SPLINE
SPL {X  -153.420, Y  +337.122, Z    +0.000, E1  +333.501, E3 -305002.639}
SPL {X  -157.288, Y  +353.220, Z    +0.000, E1  +341.134, E3 -305014.684}
SPL {X  -159.049, Y  +365.172, Z    +0.000, E1  +347.392, E3 -305020.238}
SPL {X  -159.749, Y  +373.719, Z    +0.000, E1  +352.250, E3 -305022.858}
SPL {X  -159.988, Y  +381.741, Z    +0.000, E1  +357.172, E3 -305024.333}
SPL {X  -159.990, Y  +387.352, Z    +0.000, E1  +361.387, E3 -305025.035}
SPL {X  -159.990, Y  +391.188, Z    +0.000, E1  +365.082, E3 -305025.576}
SPL {X  -159.990, Y  +395.106, Z    +0.000, E1  +369.154, E3 -305026.317}
SPL {X  -159.990, Y  +400.303, Z    +0.000, E1  +374.927, E3 -305027.638}
SPL {X  -159.990, Y  +408.423, Z    +0.000, E1  +383.302, E3 -305030.717}
SPL {X  -159.990, Y  +438.418, Z    +0.000, E1  +401.067, E3 -305052.290}
SPL {X  -159.990, Y  +482.913, Z    +0.000, E1  +407.036, E3 -305111.644}
SPL {X  -159.990, Y  +489.230, Z    +0.000, E1  +407.019, E3 -305124.156}
SPL {X  -159.990, Y  +495.241, Z    +0.000, E1  +407.026, E3 -305136.035}
SPL {X  -159.990, Y  +501.001, Z    +0.000, E1  +407.020, E3 -305147.412}
SPL {X  -159.990, Y  +506.758, Z    +0.000, E1  +407.038, E3 -305158.758}
SPL {X  -159.990, Y  +512.807, Z    +0.000, E1  +407.022, E3 -305170.749}
SPL {X  -159.990, Y  +518.043, Z    +0.000, E1  +407.016, E3 -305181.127}
SPL {X  -159.990, Y  +523.058, Z    +0.000, E1  +407.015, E3 -305191.042}
SPL {X  -159.990, Y  +527.746, Z    +0.000, E1  +407.012, E3 -305200.316}
SPL {X  -159.990, Y  +533.771, Z    +0.000, E1  +407.034, E3 -305212.201}
SPL {X  -159.990, Y  +542.379, Z    +0.000, E1  +407.067, E3 -305229.170}
SPL {X  -159.990, Y  +549.846, Z    +0.000, E1  +407.016, E3 -305244.016}
SPL {X  -159.990, Y  +554.843, Z    +0.000, E1  +407.014, E3 -305253.894}
SPL {X  -159.990, Y  +560.453, Z    +0.000, E1  +407.023, E3 -305264.977}
SPL {X  -159.990, Y  +566.612, Z    +0.000, E1  +407.022, E3 -305277.159}
SPL {X  -159.990, Y  +572.901, Z    +0.000, E1  +407.028, E3 -305289.571}
SPL {X  -159.990, Y  +578.640, Z    +0.000, E1  +407.021, E3 -305300.922}
SPL {X  -159.990, Y  +583.515, Z    +0.000, E1  +407.019, E3 -305310.562}
SPL {X  -159.990, Y  +589.675, Z    +0.000, E1  +407.042, E3 -305322.700}
SPL {X  -159.990, Y  +596.627, Z    +0.000, E1  +407.034, E3 -305336.440}
SPL {X  -159.990, Y  +602.039, Z    +0.000, E1  +407.021, E3 -305347.147}
SPL {X  -159.990, Y  +607.106, Z    +0.000, E1  +407.028, E3 -305357.154}
SPL {X  -159.990, Y  +612.418, Z    +0.000, E1  +407.023, E3 -305367.665}
SPL {X  -159.990, Y  +618.496, Z    +0.000, E1  +407.049, E3 -305379.632}
SPL {X  -159.990, Y  +624.357, Z    +0.000, E1  +407.020, E3 -305391.258}
SPL {X  -159.990, Y  +629.711, Z    +0.000, E1  +407.034, E3 -305401.827}
SPL {X  -159.990, Y  +635.041, Z    +0.000, E1  +407.022, E3 -305412.372}
SPL {X  -159.990, Y  +639.998, Z    +0.000, E1  +407.027, E3 -305422.164}
SPL {X  -159.990, Y  +646.188, Z    +0.000, E1  +407.041, E3 -305434.390}
SPL {X  -159.990, Y  +652.067, Z    +0.000, E1  +407.023, E3 -305446.026}
SPL {X  -159.990, Y  +657.109, Z    +0.000, E1  +407.025, E3 -305456.005}
SPL {X  -159.990, Y  +662.651, Z    +0.000, E1  +407.027, E3 -305466.961}
SPL {X  -159.990, Y  +668.015, Z    +0.000, E1  +407.025, E3 -305477.561}
SPL {X  -159.972, Y  +673.909, Z    +0.000, E1  +407.029, E3 -305489.226}
SPL {X  -159.776, Y  +679.772, Z    +0.000, E1  +406.992, E3 -305501.027}
SPL {X  -159.384, Y  +685.411, Z    +0.000, E1  +406.921, E3 -305512.589}
SPL {X  -158.839, Y  +690.657, Z    +0.000, E1  +406.819, E3 -305523.543}
SPL {X  -157.875, Y  +697.431, Z    +0.000, E1  +406.688, E3 -305537.882}
SPL {X  -156.719, Y  +703.686, Z    +0.000, E1  +406.438, E3 -305551.492}
SPL {X  -155.778, Y  +707.970, Z    +0.000, E1  +406.262, E3 -305560.966}
SPL {X  -154.419, Y  +713.351, Z    +0.000, E1  +406.025, E3 -305572.998}
SPL {X  -152.913, Y  +718.557, Z    +0.000, E1  +405.729, E3 -305584.850}
SPL {X  -151.262, Y  +723.621, Z    +0.000, E1  +405.429, E3 -305596.516}
SPL {X  -149.074, Y  +729.584, Z    +0.000, E1  +405.040, E3 -305610.445}
SPL {X  -142.577, Y  +744.086, Z    +0.000, E1  +400.686, E3 -305676.651}
ENDSPLINE

SPLINE
SPL {X  -152.566, Y  +719.671, Z    +0.000, E1  +387.682, E3 -305747.122}
SPL {X  -158.253, Y  +695.011, Z    +0.000, E1  +375.913, E3 -305763.793}
SPL {X  -159.486, Y  +684.192, Z    +0.000, E1  +369.965, E3 -305767.740}
SPL {X  -159.898, Y  +676.924, Z    +0.000, E1  +365.683, E3 -305769.438}
SPL {X  -159.990, Y  +671.720, Z    +0.000, E1  +362.298, E3 -305770.278}
SPL {X  -159.990, Y  +668.164, Z    +0.000, E1  +359.695, E3 -305770.693}
SPL {X  -159.990, Y  +665.062, Z    +0.000, E1  +356.961, E3 -305771.033}
SPL {X  -159.990, Y  +660.795, Z    +0.000, E1  +352.651, E3 -305771.696}
SPL {X  -159.990, Y  +654.574, Z    +0.000, E1  +345.673, E3 -305773.151}
SPL {X  -159.990, Y  +647.816, Z    +0.000, E1  +338.252, E3 -305775.402}
SPL {X  -159.990, Y  +640.751, Z    +0.000, E1  +331.747, E3 -305778.996}
SPL {X  -159.990, Y  +611.706, Z    +0.000, E1  +317.244, E3 -305801.769}
SPL {X  -159.990, Y  +567.814, Z    +0.000, E1  +312.360, E3 -305861.859}
SPL {X  -159.990, Y  +558.774, Z    +0.000, E1  +312.384, E3 -305879.424}
SPL {X  -159.990, Y  +550.551, Z    +0.000, E1  +312.385, E3 -305895.365}
SPL {X  -159.990, Y  +542.502, Z    +0.000, E1  +312.392, E3 -305910.980}
SPL {X  -159.990, Y  +536.986, Z    +0.000, E1  +312.423, E3 -305921.701}
SPL {X  -159.990, Y  +532.938, Z    +0.000, E1  +312.415, E3 -305929.527}
SPL {X  -159.990, Y  +525.893, Z    +0.000, E1  +312.375, E3 -305943.141}
SPL {X  -159.990, Y  +518.864, Z    +0.000, E1  +312.415, E3 -305956.823}
SPL {X  -159.990, Y  +512.328, Z    +0.000, E1  +312.388, E3 -305969.457}
SPL {X  -159.990, Y  +505.755, Z    +0.000, E1  +312.413, E3 -305982.234}
ENDSPLINE

SPLINE
SPL {X  -159.990, Y  +517.758, Z    +0.000, E1  +318.109, E3 -305989.957}
ENDSPLINE

SPLINE
SPL {X  -159.990, Y  +516.975, Z    +0.000, E1  +319.588, E3 -306001.020}
SPL {X  -159.990, Y  +508.583, Z    +0.000, E1  +318.552, E3 -306015.326}
SPL {X  -159.990, Y  +499.983, Z    +0.000, E1  +317.561, E3 -306029.780}
SPL {X  -159.990, Y  +492.624, Z    +0.000, E1  +316.776, E3 -306041.884}
SPL {X  -159.990, Y  +485.551, Z    +0.000, E1  +316.053, E3 -306053.433}
SPL {X  -159.990, Y  +477.585, Z    +0.000, E1  +315.156, E3 -306065.344}
SPL {X  -159.990, Y  +470.785, Z    +0.000, E1  +314.453, E3 -306075.517}
SPL {X  -159.990, Y  +463.371, Z    +0.000, E1  +313.690, E3 -306086.242}
SPL {X  -159.990, Y  +455.469, Z    +0.000, E1  +312.807, E3 -306096.768}
SPL {X  -159.990, Y  +445.848, Z    +0.000, E1  +311.866, E3 -306109.860}
SPL {X  -159.990, Y  +436.400, Z    +0.000, E1  +311.449, E3 -306125.242}
SPL {X  -159.990, Y  +429.614, Z    +0.000, E1  +311.486, E3 -306138.032}
SPL {X  -159.990, Y  +423.677, Z    +0.000, E1  +311.471, E3 -306149.144}
SPL {X  -159.990, Y  +417.714, Z    +0.000, E1  +311.484, E3 -306160.354}
SPL {X  -159.990, Y  +412.449, Z    +0.000, E1  +311.483, E3 -306170.214}
SPL {X  -159.990, Y  +406.256, Z    +0.000, E1  +311.459, E3 -306181.782}
SPL {X  -159.990, Y  +399.971, Z    +0.000, E1  +311.480, E3 -306193.597}
SPL {X  -159.990, Y  +394.711, Z    +0.000, E1  +311.476, E3 -306203.455}
SPL {X  -159.990, Y  +387.710, Z    +0.000, E1  +311.455, E3 -306216.578}
SPL {X  -159.966, Y  +379.751, Z    +0.000, E1  +311.465, E3 -306231.542}
SPL {X  -159.734, Y  +373.449, Z    +0.000, E1  +311.528, E3 -306243.646}
SPL {X  -159.230, Y  +366.920, Z    +0.000, E1  +311.592, E3 -306256.389}
SPL {X  -158.532, Y  +360.951, Z    +0.000, E1  +311.745, E3 -306268.363}
SPL {X  -157.692, Y  +355.479, Z    +0.000, E1  +311.882, E3 -306279.491}
SPL {X  -156.349, Y  +348.560, Z    +0.000, E1  +312.101, E3 -306293.830}
SPL {X  -154.984, Y  +342.790, Z    +0.000, E1  +312.392, E3 -306306.127}
SPL {X  -153.247, Y  +336.540, Z    +0.000, E1  +312.660, E3 -306319.562}
SPL {X  -150.765, Y  +328.959, Z    +0.000, E1  +313.136, E3 -306336.309}
SPL {X  -148.834, Y  +323.804, Z    +0.000, E1  +313.556, E3 -306347.962}
SPL {X  -147.343, Y  +320.157, Z    +0.000, E1  +313.838, E3 -306356.251}
SPL {X  -142.380, Y  +309.529, Z    +0.000, E1  +319.953, E3 -306429.012}
ENDSPLINE

SPLINE
SPL {X  -153.420, Y  +337.122, Z    +0.000, E1  +333.501, E3 -306486.510}
SPL {X  -157.288, Y  +353.220, Z    +0.000, E1  +341.134, E3 -306498.555}
SPL {X  -159.049, Y  +365.172, Z    +0.000, E1  +347.392, E3 -306504.109}
SPL {X  -159.749, Y  +373.719, Z    +0.000, E1  +352.250, E3 -306506.729}
SPL {X  -159.988, Y  +381.741, Z    +0.000, E1  +357.172, E3 -306508.204}
SPL {X  -159.990, Y  +387.352, Z    +0.000, E1  +361.387, E3 -306508.906}
SPL {X  -159.990, Y  +391.188, Z    +0.000, E1  +365.082, E3 -306509.447}
SPL {X  -159.990, Y  +395.106, Z    +0.000, E1  +369.154, E3 -306510.188}
SPL {X  -159.990, Y  +400.303, Z    +0.000, E1  +374.927, E3 -306511.509}
SPL {X  -159.990, Y  +408.423, Z    +0.000, E1  +383.302, E3 -306514.588}
SPL {X  -159.990, Y  +438.418, Z    +0.000, E1  +401.067, E3 -306536.161}
SPL {X  -159.990, Y  +482.913, Z    +0.000, E1  +407.036, E3 -306595.515}
SPL {X  -159.990, Y  +489.230, Z    +0.000, E1  +407.019, E3 -306608.027}
SPL {X  -159.990, Y  +495.241, Z    +0.000, E1  +407.026, E3 -306619.906}
SPL {X  -159.990, Y  +501.001, Z    +0.000, E1  +407.020, E3 -306631.283}
SPL {X  -159.990, Y  +506.758, Z    +0.000, E1  +407.038, E3 -306642.629}
SPL {X  -159.990, Y  +512.807, Z    +0.000, E1  +407.022, E3 -306654.620}
SPL {X  -159.990, Y  +518.043, Z    +0.000, E1  +407.016, E3 -306664.998}
SPL {X  -159.990, Y  +523.058, Z    +0.000, E1  +407.015, E3 -306674.913}
SPL {X  -159.990, Y  +527.746, Z    +0.000, E1  +407.012, E3 -306684.187}
SPL {X  -159.990, Y  +533.771, Z    +0.000, E1  +407.034, E3 -306696.072}
SPL {X  -159.990, Y  +542.379, Z    +0.000, E1  +407.067, E3 -306713.041}
SPL {X  -159.990, Y  +549.846, Z    +0.000, E1  +407.016, E3 -306727.887}
SPL {X  -159.990, Y  +554.843, Z    +0.000, E1  +407.014, E3 -306737.765}
SPL {X  -159.990, Y  +560.453, Z    +0.000, E1  +407.023, E3 -306748.848}
SPL {X  -159.990, Y  +566.612, Z    +0.000, E1  +407.022, E3 -306761.030}
SPL {X  -159.990, Y  +572.901, Z    +0.000, E1  +407.028, E3 -306773.442}
SPL {X  -159.990, Y  +578.640, Z    +0.000, E1  +407.021, E3 -306784.793}
SPL {X  -159.990, Y  +583.515, Z    +0.000, E1  +407.019, E3 -306794.433}
SPL {X  -159.990, Y  +589.675, Z    +0.000, E1  +407.042, E3 -306806.571}
SPL {X  -159.990, Y  +596.627, Z    +0.000, E1  +407.034, E3 -306820.311}
SPL {X  -159.990, Y  +602.039, Z    +0.000, E1  +407.021, E3 -306831.018}
SPL {X  -159.990, Y  +607.106, Z    +0.000, E1  +407.028, E3 -306841.025}
SPL {X  -159.990, Y  +612.418, Z    +0.000, E1  +407.023, E3 -306851.536}
SPL {X  -159.990, Y  +618.496, Z    +0.000, E1  +407.049, E3 -306863.503}
SPL {X  -159.990, Y  +624.357, Z    +0.000, E1  +407.020, E3 -306875.129}
SPL {X  -159.990, Y  +629.711, Z    +0.000, E1  +407.034, E3 -306885.698}
SPL {X  -159.990, Y  +635.041, Z    +0.000, E1  +407.022, E3 -306896.243}
SPL {X  -159.990, Y  +639.998, Z    +0.000, E1  +407.027, E3 -306906.035}
SPL {X  -159.990, Y  +646.188, Z    +0.000, E1  +407.041, E3 -306918.261}
SPL {X  -159.990, Y  +652.067, Z    +0.000, E1  +407.023, E3 -306929.897}
SPL {X  -159.990, Y  +657.109, Z    +0.000, E1  +407.025, E3 -306939.876}
SPL {X  -159.990, Y  +662.651, Z    +0.000, E1  +407.027, E3 -306950.832}
SPL {X  -159.990, Y  +668.015, Z    +0.000, E1  +407.025, E3 -306961.432}
SPL {X  -159.972, Y  +673.909, Z    +0.000, E1  +407.029, E3 -306973.097}
SPL {X  -159.776, Y  +679.772, Z    +0.000, E1  +406.992, E3 -306984.898}
SPL {X  -159.384, Y  +685.411, Z    +0.000, E1  +406.921, E3 -306996.460}
SPL {X  -158.839, Y  +690.657, Z    +0.000, E1  +406.819, E3 -307007.414}
SPL {X  -157.875, Y  +697.431, Z    +0.000, E1  +406.688, E3 -307021.753}
SPL {X  -156.719, Y  +703.686, Z    +0.000, E1  +406.438, E3 -307035.362}
SPL {X  -155.778, Y  +707.970, Z    +0.000, E1  +406.262, E3 -307044.837}
SPL {X  -154.419, Y  +713.351, Z    +0.000, E1  +406.025, E3 -307056.869}
SPL {X  -152.913, Y  +718.557, Z    +0.000, E1  +405.729, E3 -307068.721}
SPL {X  -151.262, Y  +723.621, Z    +0.000, E1  +405.429, E3 -307080.387}
SPL {X  -149.074, Y  +729.584, Z    +0.000, E1  +405.040, E3 -307094.316}
SPL {X  -142.577, Y  +744.086, Z    +0.000, E1  +400.686, E3 -307160.522}
ENDSPLINE

SPLINE
SPL {X  -152.566, Y  +719.671, Z    +0.000, E1  +387.682, E3 -307230.993}
SPL {X  -158.253, Y  +695.011, Z    +0.000, E1  +375.913, E3 -307247.664}
SPL {X  -159.486, Y  +684.192, Z    +0.000, E1  +369.965, E3 -307251.611}
SPL {X  -159.898, Y  +676.924, Z    +0.000, E1  +365.683, E3 -307253.309}
SPL {X  -159.990, Y  +671.720, Z    +0.000, E1  +362.298, E3 -307254.149}
SPL {X  -159.990, Y  +668.164, Z    +0.000, E1  +359.695, E3 -307254.564}
SPL {X  -159.990, Y  +665.062, Z    +0.000, E1  +356.961, E3 -307254.904}
SPL {X  -159.990, Y  +660.795, Z    +0.000, E1  +352.651, E3 -307255.567}
SPL {X  -159.990, Y  +654.574, Z    +0.000, E1  +345.673, E3 -307257.022}
SPL {X  -159.990, Y  +647.816, Z    +0.000, E1  +338.252, E3 -307259.273}
SPL {X  -159.990, Y  +640.751, Z    +0.000, E1  +331.747, E3 -307262.867}
SPL {X  -159.990, Y  +611.706, Z    +0.000, E1  +317.244, E3 -307285.640}
SPL {X  -159.990, Y  +567.814, Z    +0.000, E1  +312.360, E3 -307345.730}
SPL {X  -159.990, Y  +558.774, Z    +0.000, E1  +312.384, E3 -307363.295}
SPL {X  -159.990, Y  +550.551, Z    +0.000, E1  +312.385, E3 -307379.236}
SPL {X  -159.990, Y  +542.502, Z    +0.000, E1  +312.392, E3 -307394.851}
SPL {X  -159.990, Y  +536.986, Z    +0.000, E1  +312.423, E3 -307405.572}
SPL {X  -159.990, Y  +532.938, Z    +0.000, E1  +312.415, E3 -307413.398}
SPL {X  -159.990, Y  +525.893, Z    +0.000, E1  +312.375, E3 -307427.012}
SPL {X  -159.990, Y  +518.864, Z    +0.000, E1  +312.415, E3 -307440.694}
SPL {X  -159.990, Y  +512.328, Z    +0.000, E1  +312.388, E3 -307453.328}
SPL {X  -159.990, Y  +505.755, Z    +0.000, E1  +312.413, E3 -307466.105}
ENDSPLINE

SPLINE
SPL {X  -159.990, Y  +517.758, Z    +0.000, E1  +318.109, E3 -307473.828}
ENDSPLINE

SPLINE
SPL {X  -159.990, Y  +516.975, Z    +0.000, E1  +319.588, E3 -307484.891}
SPL {X  -159.990, Y  +508.583, Z    +0.000, E1  +318.552, E3 -307499.197}
SPL {X  -159.990, Y  +499.983, Z    +0.000, E1  +317.561, E3 -307513.651}
SPL {X  -159.990, Y  +492.624, Z    +0.000, E1  +316.776, E3 -307525.755}
SPL {X  -159.990, Y  +485.551, Z    +0.000, E1  +316.053, E3 -307537.304}
SPL {X  -159.990, Y  +477.585, Z    +0.000, E1  +315.156, E3 -307549.215}
SPL {X  -159.990, Y  +470.785, Z    +0.000, E1  +314.453, E3 -307559.388}
SPL {X  -159.990, Y  +463.371, Z    +0.000, E1  +313.690, E3 -307570.113}
SPL {X  -159.990, Y  +455.469, Z    +0.000, E1  +312.807, E3 -307580.639}
SPL {X  -159.990, Y  +445.848, Z    +0.000, E1  +311.866, E3 -307593.731}
SPL {X  -159.990, Y  +436.400, Z    +0.000, E1  +311.449, E3 -307609.113}
SPL {X  -159.990, Y  +429.614, Z    +0.000, E1  +311.486, E3 -307621.903}
SPL {X  -159.990, Y  +423.677, Z    +0.000, E1  +311.471, E3 -307633.015}
SPL {X  -159.990, Y  +417.714, Z    +0.000, E1  +311.484, E3 -307644.225}
SPL {X  -159.990, Y  +412.449, Z    +0.000, E1  +311.483, E3 -307654.085}
SPL {X  -159.990, Y  +406.256, Z    +0.000, E1  +311.459, E3 -307665.653}
SPL {X  -159.990, Y  +399.971, Z    +0.000, E1  +311.480, E3 -307677.467}
SPL {X  -159.990, Y  +394.711, Z    +0.000, E1  +311.476, E3 -307687.326}
SPL {X  -159.990, Y  +387.710, Z    +0.000, E1  +311.455, E3 -307700.449}
SPL {X  -159.966, Y  +379.751, Z    +0.000, E1  +311.465, E3 -307715.413}
SPL {X  -159.734, Y  +373.449, Z    +0.000, E1  +311.528, E3 -307727.517}
SPL {X  -159.230, Y  +366.920, Z    +0.000, E1  +311.592, E3 -307740.260}
SPL {X  -158.532, Y  +360.951, Z    +0.000, E1  +311.745, E3 -307752.234}
SPL {X  -157.692, Y  +355.479, Z    +0.000, E1  +311.882, E3 -307763.362}
SPL {X  -156.349, Y  +348.560, Z    +0.000, E1  +312.101, E3 -307777.701}
SPL {X  -154.984, Y  +342.790, Z    +0.000, E1  +312.392, E3 -307789.998}
SPL {X  -153.247, Y  +336.540, Z    +0.000, E1  +312.660, E3 -307803.433}
SPL {X  -150.765, Y  +328.959, Z    +0.000, E1  +313.136, E3 -307820.180}
SPL {X  -148.834, Y  +323.804, Z    +0.000, E1  +313.556, E3 -307831.833}
SPL {X  -147.343, Y  +320.157, Z    +0.000, E1  +313.838, E3 -307840.122}
SPL {X  -142.380, Y  +309.529, Z    +0.000, E1  +319.953, E3 -307912.883}
ENDSPLINE

SPLINE
SPL {X  -153.420, Y  +337.122, Z    +0.000, E1  +333.501, E3 -307970.381}
SPL {X  -157.288, Y  +353.220, Z    +0.000, E1  +341.134, E3 -307982.426}
SPL {X  -159.049, Y  +365.172, Z    +0.000, E1  +347.392, E3 -307987.980}
SPL {X  -159.749, Y  +373.719, Z    +0.000, E1  +352.250, E3 -307990.600}
SPL {X  -159.988, Y  +381.741, Z    +0.000, E1  +357.172, E3 -307992.075}
SPL {X  -159.990, Y  +387.352, Z    +0.000, E1  +361.387, E3 -307992.777}
SPL {X  -159.990, Y  +391.188, Z    +0.000, E1  +365.082, E3 -307993.318}
SPL {X  -159.990, Y  +395.106, Z    +0.000, E1  +369.154, E3 -307994.059}
SPL {X  -159.990, Y  +400.303, Z    +0.000, E1  +374.927, E3 -307995.380}
SPL {X  -159.990, Y  +408.423, Z    +0.000, E1  +383.302, E3 -307998.459}
SPL {X  -159.990, Y  +438.418, Z    +0.000, E1  +401.067, E3 -308020.032}
SPL {X  -159.990, Y  +482.913, Z    +0.000, E1  +407.036, E3 -308079.386}
SPL {X  -159.990, Y  +489.230, Z    +0.000, E1  +407.019, E3 -308091.898}
SPL {X  -159.990, Y  +495.241, Z    +0.000, E1  +407.026, E3 -308103.777}
SPL {X  -159.990, Y  +501.001, Z    +0.000, E1  +407.020, E3 -308115.154}
SPL {X  -159.990, Y  +506.758, Z    +0.000, E1  +407.038, E3 -308126.500}
SPL {X  -159.990, Y  +512.807, Z    +0.000, E1  +407.022, E3 -308138.491}
SPL {X  -159.990, Y  +518.043, Z    +0.000, E1  +407.016, E3 -308148.869}
SPL {X  -159.990, Y  +523.058, Z    +0.000, E1  +407.015, E3 -308158.784}
SPL {X  -159.990, Y  +527.746, Z    +0.000, E1  +407.012, E3 -308168.058}
SPL {X  -159.990, Y  +533.771, Z    +0.000, E1  +407.034, E3 -308179.943}
SPL {X  -159.990, Y  +542.379, Z    +0.000, E1  +407.067, E3 -308196.912}
SPL {X  -159.990, Y  +549.846, Z    +0.000, E1  +407.016, E3 -308211.758}
SPL {X  -159.990, Y  +554.843, Z    +0.000, E1  +407.014, E3 -308221.636}
SPL {X  -159.990, Y  +560.453, Z    +0.000, E1  +407.023, E3 -308232.719}
SPL {X  -159.990, Y  +566.612, Z    +0.000, E1  +407.022, E3 -308244.901}
SPL {X  -159.990, Y  +572.901, Z    +0.000, E1  +407.028, E3 -308257.313}
SPL {X  -159.990, Y  +578.640, Z    +0.000, E1  +407.021, E3 -308268.664}
SPL {X  -159.990, Y  +583.515, Z    +0.000, E1  +407.019, E3 -308278.304}
SPL {X  -159.990, Y  +589.675, Z    +0.000, E1  +407.042, E3 -308290.442}
SPL {X  -159.990, Y  +596.627, Z    +0.000, E1  +407.034, E3 -308304.182}
SPL {X  -159.990, Y  +602.039, Z    +0.000, E1  +407.021, E3 -308314.889}
SPL {X  -159.990, Y  +607.106, Z    +0.000, E1  +407.028, E3 -308324.896}
SPL {X  -159.990, Y  +612.418, Z    +0.000, E1  +407.023, E3 -308335.407}
SPL {X  -159.990, Y  +618.496, Z    +0.000, E1  +407.049, E3 -308347.374}
SPL {X  -159.990, Y  +624.357, Z    +0.000, E1  +407.020, E3 -308359.000}
SPL {X  -159.990, Y  +629.711, Z    +0.000, E1  +407.034, E3 -308369.569}
SPL {X  -159.990, Y  +635.041, Z    +0.000, E1  +407.022, E3 -308380.114}
SPL {X  -159.990, Y  +639.998, Z    +0.000, E1  +407.027, E3 -308389.906}
SPL {X  -159.990, Y  +646.188, Z    +0.000, E1  +407.041, E3 -308402.132}
SPL {X  -159.990, Y  +652.067, Z    +0.000, E1  +407.023, E3 -308413.768}
SPL {X  -159.990, Y  +657.109, Z    +0.000, E1  +407.025, E3 -308423.747}
SPL {X  -159.990, Y  +662.651, Z    +0.000, E1  +407.027, E3 -308434.703}
SPL {X  -159.990, Y  +668.015, Z    +0.000, E1  +407.025, E3 -308445.303}
SPL {X  -159.972, Y  +673.909, Z    +0.000, E1  +407.029, E3 -308456.968}
SPL {X  -159.776, Y  +679.772, Z    +0.000, E1  +406.992, E3 -308468.769}
SPL {X  -159.384, Y  +685.411, Z    +0.000, E1  +406.921, E3 -308480.331}
SPL {X  -158.839, Y  +690.657, Z    +0.000, E1  +406.819, E3 -308491.285}
SPL {X  -157.875, Y  +697.431, Z    +0.000, E1  +406.688, E3 -308505.624}
SPL {X  -156.719, Y  +703.686, Z    +0.000, E1  +406.438, E3 -308519.233}
SPL {X  -155.778, Y  +707.970, Z    +0.000, E1  +406.262, E3 -308528.708}
SPL {X  -154.419, Y  +713.351, Z    +0.000, E1  +406.025, E3 -308540.740}
SPL {X  -152.913, Y  +718.557, Z    +0.000, E1  +405.729, E3 -308552.592}
SPL {X  -151.262, Y  +723.621, Z    +0.000, E1  +405.429, E3 -308564.258}
SPL {X  -149.074, Y  +729.584, Z    +0.000, E1  +405.040, E3 -308578.187}
SPL {X  -142.577, Y  +744.086, Z    +0.000, E1  +400.686, E3 -308644.393}
ENDSPLINE

SPLINE
SPL {X  -152.566, Y  +719.671, Z    +0.000, E1  +387.682, E3 -308714.864}
SPL {X  -158.253, Y  +695.011, Z    +0.000, E1  +375.913, E3 -308731.535}
SPL {X  -159.486, Y  +684.192, Z    +0.000, E1  +369.965, E3 -308735.482}
SPL {X  -159.898, Y  +676.924, Z    +0.000, E1  +365.683, E3 -308737.180}
SPL {X  -159.990, Y  +671.720, Z    +0.000, E1  +362.298, E3 -308738.020}
SPL {X  -159.990, Y  +668.164, Z    +0.000, E1  +359.695, E3 -308738.435}
SPL {X  -159.990, Y  +665.062, Z    +0.000, E1  +356.961, E3 -308738.775}
SPL {X  -159.990, Y  +660.795, Z    +0.000, E1  +352.651, E3 -308739.438}
SPL {X  -159.990, Y  +654.574, Z    +0.000, E1  +345.673, E3 -308740.893}
SPL {X  -159.990, Y  +647.816, Z    +0.000, E1  +338.252, E3 -308743.144}
SPL {X  -159.990, Y  +640.751, Z    +0.000, E1  +331.747, E3 -308746.738}
SPL {X  -159.990, Y  +611.706, Z    +0.000, E1  +317.244, E3 -308769.511}
SPL {X  -159.990, Y  +567.814, Z    +0.000, E1  +312.360, E3 -308829.601}
SPL {X  -159.990, Y  +558.774, Z    +0.000, E1  +312.384, E3 -308847.166}
SPL {X  -159.990, Y  +550.551, Z    +0.000, E1  +312.385, E3 -308863.107}
SPL {X  -159.990, Y  +542.502, Z    +0.000, E1  +312.392, E3 -308878.722}
SPL {X  -159.990, Y  +536.986, Z    +0.000, E1  +312.423, E3 -308889.443}
SPL {X  -159.990, Y  +532.938, Z    +0.000, E1  +312.415, E3 -308897.269}
SPL {X  -159.990, Y  +525.893, Z    +0.000, E1  +312.375, E3 -308910.883}
SPL {X  -159.990, Y  +518.864, Z    +0.000, E1  +312.415, E3 -308924.565}
SPL {X  -159.990, Y  +512.328, Z    +0.000, E1  +312.388, E3 -308937.199}
SPL {X  -159.990, Y  +505.755, Z    +0.000, E1  +312.413, E3 -308949.976}
ENDSPLINE

SPLINE
SPL {X  -159.990, Y  +517.758, Z    +0.000, E1  +318.109, E3 -308957.699}
ENDSPLINE

SPLINE
SPL {X  -159.990, Y  +516.975, Z    +0.000, E1  +319.588, E3 -308968.762}
SPL {X  -159.990, Y  +508.583, Z    +0.000, E1  +318.552, E3 -308983.068}
SPL {X  -159.990, Y  +499.983, Z    +0.000, E1  +317.561, E3 -308997.522}
SPL {X  -159.990, Y  +492.624, Z    +0.000, E1  +316.776, E3 -309009.626}
SPL {X  -159.990, Y  +485.551, Z    +0.000, E1  +316.053, E3 -309021.175}
SPL {X  -159.990, Y  +477.585, Z    +0.000, E1  +315.156, E3 -309033.086}
SPL {X  -159.990, Y  +470.785, Z    +0.000, E1  +314.453, E3 -309043.259}
SPL {X  -159.990, Y  +463.371, Z    +0.000, E1  +313.690, E3 -309053.984}
SPL {X  -159.990, Y  +455.469, Z    +0.000, E1  +312.807, E3 -309064.510}
SPL {X  -159.990, Y  +445.848, Z    +0.000, E1  +311.866, E3 -309077.602}
SPL {X  -159.990, Y  +436.400, Z    +0.000, E1  +311.449, E3 -309092.984}
SPL {X  -159.990, Y  +429.614, Z    +0.000, E1  +311.486, E3 -309105.774}
SPL {X  -159.990, Y  +423.677, Z    +0.000, E1  +311.471, E3 -309116.886}
SPL {X  -159.990, Y  +417.714, Z    +0.000, E1  +311.484, E3 -309128.096}
SPL {X  -159.990, Y  +412.449, Z    +0.000, E1  +311.483, E3 -309137.956}
SPL {X  -159.990, Y  +406.256, Z    +0.000, E1  +311.459, E3 -309149.524}
SPL {X  -159.990, Y  +399.971, Z    +0.000, E1  +311.480, E3 -309161.338}
SPL {X  -159.990, Y  +394.711, Z    +0.000, E1  +311.476, E3 -309171.197}
SPL {X  -159.990, Y  +387.710, Z    +0.000, E1  +311.455, E3 -309184.320}
SPL {X  -159.966, Y  +379.751, Z    +0.000, E1  +311.465, E3 -309199.284}
SPL {X  -159.734, Y  +373.449, Z    +0.000, E1  +311.528, E3 -309211.388}
SPL {X  -159.230, Y  +366.920, Z    +0.000, E1  +311.592, E3 -309224.131}
SPL {X  -158.532, Y  +360.951, Z    +0.000, E1  +311.745, E3 -309236.105}
SPL {X  -157.692, Y  +355.479, Z    +0.000, E1  +311.882, E3 -309247.233}
SPL {X  -156.349, Y  +348.560, Z    +0.000, E1  +312.101, E3 -309261.572}
SPL {X  -154.984, Y  +342.790, Z    +0.000, E1  +312.392, E3 -309273.869}
SPL {X  -153.247, Y  +336.540, Z    +0.000, E1  +312.660, E3 -309287.304}
SPL {X  -150.765, Y  +328.959, Z    +0.000, E1  +313.136, E3 -309304.051}
SPL {X  -148.834, Y  +323.804, Z    +0.000, E1  +313.556, E3 -309315.704}
SPL {X  -147.343, Y  +320.157, Z    +0.000, E1  +313.838, E3 -309323.993}
SPL {X  -142.380, Y  +309.529, Z    +0.000, E1  +319.953, E3 -309396.754}
ENDSPLINE

SPLINE
SPL {X  -153.420, Y  +337.122, Z    +0.000, E1  +333.501, E3 -309454.252}
SPL {X  -157.288, Y  +353.220, Z    +0.000, E1  +341.134, E3 -309466.297}
SPL {X  -159.049, Y  +365.172, Z    +0.000, E1  +347.392, E3 -309471.851}
SPL {X  -159.749, Y  +373.719, Z    +0.000, E1  +352.250, E3 -309474.471}
SPL {X  -159.988, Y  +381.741, Z    +0.000, E1  +357.172, E3 -309475.946}
SPL {X  -159.990, Y  +387.352, Z    +0.000, E1  +361.387, E3 -309476.648}
SPL {X  -159.990, Y  +391.188, Z    +0.000, E1  +365.082, E3 -309477.189}
SPL {X  -159.990, Y  +395.106, Z    +0.000, E1  +369.154, E3 -309477.930}
SPL {X  -159.990, Y  +400.303, Z    +0.000, E1  +374.927, E3 -309479.251}
SPL {X  -159.990, Y  +408.423, Z    +0.000, E1  +383.302, E3 -309482.330}
SPL {X  -159.990, Y  +438.418, Z    +0.000, E1  +401.067, E3 -309503.903}
SPL {X  -159.990, Y  +482.913, Z    +0.000, E1  +407.036, E3 -309563.257}
SPL {X  -159.990, Y  +489.230, Z    +0.000, E1  +407.019, E3 -309575.769}
SPL {X  -159.990, Y  +495.241, Z    +0.000, E1  +407.026, E3 -309587.648}
SPL {X  -159.990, Y  +501.001, Z    +0.000, E1  +407.020, E3 -309599.025}
SPL {X  -159.990, Y  +506.758, Z    +0.000, E1  +407.038, E3 -309610.371}
SPL {X  -159.990, Y  +512.807, Z    +0.000, E1  +407.022, E3 -309622.362}
SPL {X  -159.990, Y  +518.043, Z    +0.000, E1  +407.016, E3 -309632.740}
SPL {X  -159.990, Y  +523.058, Z    +0.000, E1  +407.015, E3 -309642.655}
SPL {X  -159.990, Y  +527.746, Z    +0.000, E1  +407.012, E3 -309651.929}
SPL {X  -159.990, Y  +533.771, Z    +0.000, E1  +407.034, E3 -309663.814}
SPL {X  -159.990, Y  +542.379, Z    +0.000, E1  +407.067, E3 -309680.783}
SPL {X  -159.990, Y  +549.846, Z    +0.000, E1  +407.016, E3 -309695.629}
SPL {X  -159.990, Y  +554.843, Z    +0.000, E1  +407.014, E3 -309705.507}
SPL {X  -159.990, Y  +560.453, Z    +0.000, E1  +407.023, E3 -309716.590}
SPL {X  -159.990, Y  +566.612, Z    +0.000, E1  +407.022, E3 -309728.772}
SPL {X  -159.990, Y  +572.901, Z    +0.000, E1  +407.028, E3 -309741.184}
SPL {X  -159.990, Y  +578.640, Z    +0.000, E1  +407.021, E3 -309752.535}
SPL {X  -159.990, Y  +583.515, Z    +0.000, E1  +407.019, E3 -309762.175}
SPL {X  -159.990, Y  +589.675, Z    +0.000, E1  +407.042, E3 -309774.313}
SPL {X  -159.990, Y  +596.627, Z    +0.000, E1  +407.034, E3 -309788.053}
SPL {X  -159.990, Y  +602.039, Z    +0.000, E1  +407.021, E3 -309798.760}
SPL {X  -159.990, Y  +607.106, Z    +0.000, E1  +407.028, E3 -309808.767}
SPL {X  -159.990, Y  +612.418, Z    +0.000, E1  +407.023, E3 -309819.278}
SPL {X  -159.990, Y  +618.496, Z    +0.000, E1  +407.049, E3 -309831.245}
SPL {X  -159.990, Y  +624.357, Z    +0.000, E1  +407.020, E3 -309842.871}
SPL {X  -159.990, Y  +629.711, Z    +0.000, E1  +407.034, E3 -309853.440}
SPL {X  -159.990, Y  +635.041, Z    +0.000, E1  +407.022, E3 -309863.985}
SPL {X  -159.990, Y  +639.998, Z    +0.000, E1  +407.027, E3 -309873.777}
SPL {X  -159.990, Y  +646.188, Z    +0.000, E1  +407.041, E3 -309886.003}
SPL {X  -159.990, Y  +652.067, Z    +0.000, E1  +407.023, E3 -309897.639}
SPL {X  -159.990, Y  +657.109, Z    +0.000, E1  +407.025, E3 -309907.618}
SPL {X  -159.990, Y  +662.651, Z    +0.000, E1  +407.027, E3 -309918.574}
SPL {X  -159.990, Y  +668.015, Z    +0.000, E1  +407.025, E3 -309929.174}
SPL {X  -159.972, Y  +673.909, Z    +0.000, E1  +407.029, E3 -309940.839}
SPL {X  -159.776, Y  +679.772, Z    +0.000, E1  +406.992, E3 -309952.640}
SPL {X  -159.384, Y  +685.411, Z    +0.000, E1  +406.921, E3 -309964.202}
SPL {X  -158.839, Y  +690.657, Z    +0.000, E1  +406.819, E3 -309975.156}
SPL {X  -157.875, Y  +697.431, Z    +0.000, E1  +406.688, E3 -309989.495}
SPL {X  -156.719, Y  +703.686, Z    +0.000, E1  +406.438, E3 -310003.104}
SPL {X  -155.778, Y  +707.970, Z    +0.000, E1  +406.262, E3 -310012.579}
SPL {X  -154.419, Y  +713.351, Z    +0.000, E1  +406.025, E3 -310024.611}
SPL {X  -152.913, Y  +718.557, Z    +0.000, E1  +405.729, E3 -310036.463}
SPL {X  -151.262, Y  +723.621, Z    +0.000, E1  +405.429, E3 -310048.129}
SPL {X  -149.074, Y  +729.584, Z    +0.000, E1  +405.040, E3 -310062.058}
SPL {X  -142.577, Y  +744.086, Z    +0.000, E1  +400.686, E3 -310128.264}
ENDSPLINE

SPLINE
SPL {X  -152.566, Y  +719.671, Z    +0.000, E1  +387.682, E3 -310198.735}
SPL {X  -158.253, Y  +695.011, Z    +0.000, E1  +375.913, E3 -310215.406}
SPL {X  -159.486, Y  +684.192, Z    +0.000, E1  +369.965, E3 -310219.353}
SPL {X  -159.898, Y  +676.924, Z    +0.000, E1  +365.683, E3 -310221.051}
SPL {X  -159.990, Y  +671.720, Z    +0.000, E1  +362.298, E3 -310221.891}
SPL {X  -159.990, Y  +668.164, Z    +0.000, E1  +359.695, E3 -310222.306}
SPL {X  -159.990, Y  +665.062, Z    +0.000, E1  +356.961, E3 -310222.646}
SPL {X  -159.990, Y  +660.795, Z    +0.000, E1  +352.651, E3 -310223.309}
SPL {X  -159.990, Y  +654.574, Z    +0.000, E1  +345.673, E3 -310224.764}
SPL {X  -159.990, Y  +647.816, Z    +0.000, E1  +338.252, E3 -310227.015}
SPL {X  -159.990, Y  +640.751, Z    +0.000, E1  +331.747, E3 -310230.609}
SPL {X  -159.990, Y  +611.706, Z    +0.000, E1  +317.244, E3 -310253.382}
SPL {X  -159.990, Y  +567.814, Z    +0.000, E1  +312.360, E3 -310313.472}
SPL {X  -159.990, Y  +558.774, Z    +0.000, E1  +312.384, E3 -310331.037}
SPL {X  -159.990, Y  +550.551, Z    +0.000, E1  +312.385, E3 -310346.978}
SPL {X  -159.990, Y  +542.502, Z    +0.000, E1  +312.392, E3 -310362.593}
SPL {X  -159.990, Y  +536.986, Z    +0.000, E1  +312.423, E3 -310373.314}
SPL {X  -159.990, Y  +532.938, Z    +0.000, E1  +312.415, E3 -310381.140}
SPL {X  -159.990, Y  +525.893, Z    +0.000, E1  +312.375, E3 -310394.754}
SPL {X  -159.990, Y  +518.864, Z    +0.000, E1  +312.415, E3 -310408.436}
SPL {X  -159.990, Y  +512.328, Z    +0.000, E1  +312.388, E3 -310421.070}
SPL {X  -159.990, Y  +505.755, Z    +0.000, E1  +312.413, E3 -310433.847}
ENDSPLINE

SPLINE
SPL {X  -159.990, Y  +517.758, Z    +0.000, E1  +318.109, E3 -310441.570}
ENDSPLINE

SPLINE
SPL {X  -159.990, Y  +516.975, Z    +0.000, E1  +319.588, E3 -310452.633}
SPL {X  -159.990, Y  +508.583, Z    +0.000, E1  +318.552, E3 -310466.938}
SPL {X  -159.990, Y  +499.983, Z    +0.000, E1  +317.561, E3 -310481.393}
SPL {X  -159.990, Y  +492.624, Z    +0.000, E1  +316.776, E3 -310493.497}
SPL {X  -159.990, Y  +485.551, Z    +0.000, E1  +316.053, E3 -310505.046}
SPL {X  -159.990, Y  +477.585, Z    +0.000, E1  +315.156, E3 -310516.957}
SPL {X  -159.990, Y  +470.785, Z    +0.000, E1  +314.453, E3 -310527.130}
SPL {X  -159.990, Y  +463.371, Z    +0.000, E1  +313.690, E3 -310537.855}
SPL {X  -159.990, Y  +455.469, Z    +0.000, E1  +312.807, E3 -310548.381}
SPL {X  -159.990, Y  +445.848, Z    +0.000, E1  +311.866, E3 -310561.473}
SPL {X  -159.990, Y  +436.400, Z    +0.000, E1  +311.449, E3 -310576.854}
SPL {X  -159.990, Y  +429.614, Z    +0.000, E1  +311.486, E3 -310589.645}
SPL {X  -159.990, Y  +423.677, Z    +0.000, E1  +311.471, E3 -310600.757}
SPL {X  -159.990, Y  +417.714, Z    +0.000, E1  +311.484, E3 -310611.967}
SPL {X  -159.990, Y  +412.449, Z    +0.000, E1  +311.483, E3 -310621.827}
SPL {X  -159.990, Y  +406.256, Z    +0.000, E1  +311.459, E3 -310633.395}
SPL {X  -159.990, Y  +399.971, Z    +0.000, E1  +311.480, E3 -310645.209}
SPL {X  -159.990, Y  +394.711, Z    +0.000, E1  +311.476, E3 -310655.068}
SPL {X  -159.990, Y  +387.710, Z    +0.000, E1  +311.455, E3 -310668.191}
SPL {X  -159.966, Y  +379.751, Z    +0.000, E1  +311.465, E3 -310683.155}
SPL {X  -159.734, Y  +373.449, Z    +0.000, E1  +311.528, E3 -310695.259}
SPL {X  -159.230, Y  +366.920, Z    +0.000, E1  +311.592, E3 -310708.002}
SPL {X  -158.532, Y  +360.951, Z    +0.000, E1  +311.745, E3 -310719.976}
SPL {X  -157.692, Y  +355.479, Z    +0.000, E1  +311.882, E3 -310731.103}
SPL {X  -156.349, Y  +348.560, Z    +0.000, E1  +312.101, E3 -310745.443}
SPL {X  -154.984, Y  +342.790, Z    +0.000, E1  +312.392, E3 -310757.740}
SPL {X  -153.247, Y  +336.540, Z    +0.000, E1  +312.660, E3 -310771.175}
SPL {X  -150.765, Y  +328.959, Z    +0.000, E1  +313.136, E3 -310787.922}
SPL {X  -148.834, Y  +323.804, Z    +0.000, E1  +313.556, E3 -310799.575}
SPL {X  -147.343, Y  +320.157, Z    +0.000, E1  +313.838, E3 -310807.864}
SPL {X  -142.380, Y  +309.529, Z    +0.000, E1  +319.953, E3 -310880.625}
ENDSPLINE

SPLINE
SPL {X  -153.420, Y  +337.122, Z    +0.000, E1  +333.501, E3 -310938.123}
SPL {X  -157.288, Y  +353.220, Z    +0.000, E1  +341.134, E3 -310950.168}
SPL {X  -159.049, Y  +365.172, Z    +0.000, E1  +347.392, E3 -310955.722}
SPL {X  -159.749, Y  +373.719, Z    +0.000, E1  +352.250, E3 -310958.342}
SPL {X  -159.988, Y  +381.741, Z    +0.000, E1  +357.172, E3 -310959.817}
SPL {X  -159.990, Y  +387.352, Z    +0.000, E1  +361.387, E3 -310960.519}
SPL {X  -159.990, Y  +391.188, Z    +0.000, E1  +365.082, E3 -310961.060}
SPL {X  -159.990, Y  +395.106, Z    +0.000, E1  +369.154, E3 -310961.801}
SPL {X  -159.990, Y  +400.303, Z    +0.000, E1  +374.927, E3 -310963.122}
SPL {X  -159.990, Y  +408.423, Z    +0.000, E1  +383.302, E3 -310966.201}
SPL {X  -159.990, Y  +438.418, Z    +0.000, E1  +401.067, E3 -310987.774}
SPL {X  -159.990, Y  +482.913, Z    +0.000, E1  +407.036, E3 -311047.128}
SPL {X  -159.990, Y  +489.230, Z    +0.000, E1  +407.019, E3 -311059.640}
SPL {X  -159.990, Y  +495.241, Z    +0.000, E1  +407.026, E3 -311071.519}
SPL {X  -159.990, Y  +501.001, Z    +0.000, E1  +407.020, E3 -311082.896}
SPL {X  -159.990, Y  +506.758, Z    +0.000, E1  +407.038, E3 -311094.242}
SPL {X  -159.990, Y  +512.807, Z    +0.000, E1  +407.022, E3 -311106.233}
SPL {X  -159.990, Y  +518.043, Z    +0.000, E1  +407.016, E3 -311116.610}
SPL {X  -159.990, Y  +523.058, Z    +0.000, E1  +407.015, E3 -311126.526}
SPL {X  -159.990, Y  +527.746, Z    +0.000, E1  +407.012, E3 -311135.800}
SPL {X  -159.990, Y  +533.771, Z    +0.000, E1  +407.034, E3 -311147.685}
SPL {X  -159.990, Y  +542.379, Z    +0.000, E1  +407.067, E3 -311164.654}
SPL {X  -159.990, Y  +549.846, Z    +0.000, E1  +407.016, E3 -311179.500}
SPL {X  -159.990, Y  +554.843, Z    +0.000, E1  +407.014, E3 -311189.378}
SPL {X  -159.990, Y  +560.453, Z    +0.000, E1  +407.023, E3 -311200.461}
SPL {X  -159.990, Y  +566.612, Z    +0.000, E1  +407.022, E3 -311212.643}
SPL {X  -159.990, Y  +572.901, Z    +0.000, E1  +407.028, E3 -311225.055}
SPL {X  -159.990, Y  +578.640, Z    +0.000, E1  +407.021, E3 -311236.406}
SPL {X  -159.990, Y  +583.515, Z    +0.000, E1  +407.019, E3 -311246.046}
SPL {X  -159.990, Y  +589.675, Z    +0.000, E1  +407.042, E3 -311258.184}
SPL {X  -159.990, Y  +596.627, Z    +0.000, E1  +407.034, E3 -311271.924}
SPL {X  -159.990, Y  +602.039, Z    +0.000, E1  +407.021, E3 -311282.631}
SPL {X  -159.990, Y  +607.106, Z    +0.000, E1  +407.028, E3 -311292.638}
SPL {X  -159.990, Y  +612.418, Z    +0.000, E1  +407.023, E3 -311303.149}
SPL {X  -159.990, Y  +618.496, Z    +0.000, E1  +407.049, E3 -311315.116}
SPL {X  -159.990, Y  +624.357, Z    +0.000, E1  +407.020, E3 -311326.742}
SPL {X  -159.990, Y  +629.711, Z    +0.000, E1  +407.034, E3 -311337.311}
SPL {X  -159.990, Y  +635.041, Z    +0.000, E1  +407.022, E3 -311347.856}
SPL {X  -159.990, Y  +639.998, Z    +0.000, E1  +407.027, E3 -311357.648}
SPL {X  -159.990, Y  +646.188, Z    +0.000, E1  +407.041, E3 -311369.874}
SPL {X  -159.990, Y  +652.067, Z    +0.000, E1  +407.023, E3 -311381.510}
SPL {X  -159.990, Y  +657.109, Z    +0.000, E1  +407.025, E3 -311391.489}
SPL {X  -159.990, Y  +662.651, Z    +0.000, E1  +407.027, E3 -311402.445}
SPL {X  -159.990, Y  +668.015, Z    +0.000, E1  +407.025, E3 -311413.045}
SPL {X  -159.972, Y  +673.909, Z    +0.000, E1  +407.029, E3 -311424.710}
SPL {X  -159.776, Y  +679.772, Z    +0.000, E1  +406.992, E3 -311436.511}
SPL {X  -159.384, Y  +685.411, Z    +0.000, E1  +406.921, E3 -311448.073}
SPL {X  -158.839, Y  +690.657, Z    +0.000, E1  +406.819, E3 -311459.027}
SPL {X  -157.875, Y  +697.431, Z    +0.000, E1  +406.688, E3 -311473.366}
SPL {X  -156.719, Y  +703.686, Z    +0.000, E1  +406.438, E3 -311486.975}
SPL {X  -155.778, Y  +707.970, Z    +0.000, E1  +406.262, E3 -311496.450}
SPL {X  -154.419, Y  +713.351, Z    +0.000, E1  +406.025, E3 -311508.482}
SPL {X  -152.913, Y  +718.557, Z    +0.000, E1  +405.729, E3 -311520.334}
SPL {X  -151.262, Y  +723.621, Z    +0.000, E1  +405.429, E3 -311532.000}
SPL {X  -149.074, Y  +729.584, Z    +0.000, E1  +405.040, E3 -311545.929}
SPL {X  -142.577, Y  +744.086, Z    +0.000, E1  +400.686, E3 -311612.135}
ENDSPLINE

SPLINE
SPL {X  -152.566, Y  +719.671, Z    +0.000, E1  +387.682, E3 -311682.606}
SPL {X  -158.253, Y  +695.011, Z    +0.000, E1  +375.913, E3 -311699.277}
SPL {X  -159.486, Y  +684.192, Z    +0.000, E1  +369.965, E3 -311703.224}
SPL {X  -159.898, Y  +676.924, Z    +0.000, E1  +365.683, E3 -311704.922}
SPL {X  -159.990, Y  +671.720, Z    +0.000, E1  +362.298, E3 -311705.762}
SPL {X  -159.990, Y  +668.164, Z    +0.000, E1  +359.695, E3 -311706.177}
SPL {X  -159.990, Y  +665.062, Z    +0.000, E1  +356.961, E3 -311706.517}
SPL {X  -159.990, Y  +660.795, Z    +0.000, E1  +352.651, E3 -311707.180}
SPL {X  -159.990, Y  +654.574, Z    +0.000, E1  +345.673, E3 -311708.634}
SPL {X  -159.990, Y  +647.816, Z    +0.000, E1  +338.252, E3 -311710.886}
SPL {X  -159.990, Y  +640.751, Z    +0.000, E1  +331.747, E3 -311714.480}
SPL {X  -159.990, Y  +611.706, Z    +0.000, E1  +317.244, E3 -311737.253}
SPL {X  -159.990, Y  +567.814, Z    +0.000, E1  +312.360, E3 -311797.343}
SPL {X  -159.990, Y  +558.774, Z    +0.000, E1  +312.384, E3 -311814.908}
SPL {X  -159.990, Y  +550.551, Z    +0.000, E1  +312.385, E3 -311830.849}
SPL {X  -159.990, Y  +542.502, Z    +0.000, E1  +312.392, E3 -311846.464}
SPL {X  -159.990, Y  +536.986, Z    +0.000, E1  +312.423, E3 -311857.185}
SPL {X  -159.990, Y  +532.938, Z    +0.000, E1  +312.415, E3 -311865.011}
SPL {X  -159.990, Y  +525.893, Z    +0.000, E1  +312.375, E3 -311878.625}
SPL {X  -159.990, Y  +518.864, Z    +0.000, E1  +312.415, E3 -311892.307}
SPL {X  -159.990, Y  +512.328, Z    +0.000, E1  +312.388, E3 -311904.941}
SPL {X  -159.990, Y  +505.755, Z    +0.000, E1  +312.413, E3 -311917.718}
ENDSPLINE

SPLINE
SPL {X  -159.990, Y  +517.758, Z    +0.000, E1  +318.109, E3 -311925.441}
ENDSPLINE

SPLINE
SPL {X  -159.990, Y  +516.975, Z    +0.000, E1  +319.588, E3 -311936.504}
SPL {X  -159.990, Y  +508.583, Z    +0.000, E1  +318.552, E3 -311950.809}
SPL {X  -159.990, Y  +499.983, Z    +0.000, E1  +317.561, E3 -311965.264}
SPL {X  -159.990, Y  +492.624, Z    +0.000, E1  +316.776, E3 -311977.368}
SPL {X  -159.990, Y  +485.551, Z    +0.000, E1  +316.053, E3 -311988.917}
SPL {X  -159.990, Y  +477.585, Z    +0.000, E1  +315.156, E3 -312000.828}
SPL {X  -159.990, Y  +470.785, Z    +0.000, E1  +314.453, E3 -312011.001}
SPL {X  -159.990, Y  +463.371, Z    +0.000, E1  +313.690, E3 -312021.726}
SPL {X  -159.990, Y  +455.469, Z    +0.000, E1  +312.807, E3 -312032.252}
SPL {X  -159.990, Y  +445.848, Z    +0.000, E1  +311.866, E3 -312045.344}
SPL {X  -159.990, Y  +436.400, Z    +0.000, E1  +311.449, E3 -312060.725}
SPL {X  -159.990, Y  +429.614, Z    +0.000, E1  +311.486, E3 -312073.516}
SPL {X  -159.990, Y  +423.677, Z    +0.000, E1  +311.471, E3 -312084.628}
SPL {X  -159.990, Y  +417.714, Z    +0.000, E1  +311.484, E3 -312095.838}
SPL {X  -159.990, Y  +412.449, Z    +0.000, E1  +311.483, E3 -312105.698}
SPL {X  -159.990, Y  +406.256, Z    +0.000, E1  +311.459, E3 -312117.265}
SPL {X  -159.990, Y  +399.971, Z    +0.000, E1  +311.480, E3 -312129.080}
SPL {X  -159.990, Y  +394.711, Z    +0.000, E1  +311.476, E3 -312138.939}
SPL {X  -159.990, Y  +387.710, Z    +0.000, E1  +311.455, E3 -312152.062}
SPL {X  -159.966, Y  +379.751, Z    +0.000, E1  +311.465, E3 -312167.026}
SPL {X  -159.734, Y  +373.449, Z    +0.000, E1  +311.528, E3 -312179.130}
SPL {X  -159.230, Y  +366.920, Z    +0.000, E1  +311.592, E3 -312191.873}
SPL {X  -158.532, Y  +360.951, Z    +0.000, E1  +311.745, E3 -312203.847}
SPL {X  -157.692, Y  +355.479, Z    +0.000, E1  +311.882, E3 -312214.974}
SPL {X  -156.349, Y  +348.560, Z    +0.000, E1  +312.101, E3 -312229.314}
SPL {X  -154.984, Y  +342.790, Z    +0.000, E1  +312.392, E3 -312241.611}
SPL {X  -153.247, Y  +336.540, Z    +0.000, E1  +312.660, E3 -312255.046}
SPL {X  -150.765, Y  +328.959, Z    +0.000, E1  +313.136, E3 -312271.793}
SPL {X  -148.834, Y  +323.804, Z    +0.000, E1  +313.556, E3 -312283.445}
SPL {X  -147.343, Y  +320.157, Z    +0.000, E1  +313.838, E3 -312291.735}
SPL {X  -142.380, Y  +309.529, Z    +0.000, E1  +319.953, E3 -312364.496}
ENDSPLINE

SPLINE
SPL {X  -153.420, Y  +337.122, Z    +0.000, E1  +333.501, E3 -312421.994}
SPL {X  -157.288, Y  +353.220, Z    +0.000, E1  +341.134, E3 -312434.039}
SPL {X  -159.049, Y  +365.172, Z    +0.000, E1  +347.392, E3 -312439.593}
SPL {X  -159.749, Y  +373.719, Z    +0.000, E1  +352.250, E3 -312442.213}
SPL {X  -159.988, Y  +381.741, Z    +0.000, E1  +357.172, E3 -312443.688}
SPL {X  -159.990, Y  +387.352, Z    +0.000, E1  +361.387, E3 -312444.390}
SPL {X  -159.990, Y  +391.188, Z    +0.000, E1  +365.082, E3 -312444.931}
SPL {X  -159.990, Y  +395.106, Z    +0.000, E1  +369.154, E3 -312445.672}
SPL {X  -159.990, Y  +400.303, Z    +0.000, E1  +374.927, E3 -312446.993}
SPL {X  -159.990, Y  +408.423, Z    +0.000, E1  +383.302, E3 -312450.072}
SPL {X  -159.990, Y  +438.418, Z    +0.000, E1  +401.067, E3 -312471.645}
SPL {X  -159.990, Y  +482.913, Z    +0.000, E1  +407.036, E3 -312530.999}
SPL {X  -159.990, Y  +489.230, Z    +0.000, E1  +407.019, E3 -312543.511}
SPL {X  -159.990, Y  +495.241, Z    +0.000, E1  +407.026, E3 -312555.390}
SPL {X  -159.990, Y  +501.001, Z    +0.000, E1  +407.020, E3 -312566.767}
SPL {X  -159.990, Y  +506.758, Z    +0.000, E1  +407.038, E3 -312578.113}
SPL {X  -159.990, Y  +512.807, Z    +0.000, E1  +407.022, E3 -312590.104}
SPL {X  -159.990, Y  +518.043, Z    +0.000, E1  +407.016, E3 -312600.481}
SPL {X  -159.990, Y  +523.058, Z    +0.000, E1  +407.015, E3 -312610.397}
SPL {X  -159.990, Y  +527.746, Z    +0.000, E1  +407.012, E3 -312619.671}
SPL {X  -159.990, Y  +533.771, Z    +0.000, E1  +407.034, E3 -312631.556}
SPL {X  -159.990, Y  +542.379, Z    +0.000, E1  +407.067, E3 -312648.525}
SPL {X  -159.990, Y  +549.846, Z    +0.000, E1  +407.016, E3 -312663.371}
SPL {X  -159.990, Y  +554.843, Z    +0.000, E1  +407.014, E3 -312673.249}
SPL {X  -159.990, Y  +560.453, Z    +0.000, E1  +407.023, E3 -312684.332}
SPL {X  -159.990, Y  +566.612, Z    +0.000, E1  +407.022, E3 -312696.514}
SPL {X  -159.990, Y  +572.901, Z    +0.000, E1  +407.028, E3 -312708.926}
SPL {X  -159.990, Y  +578.640, Z    +0.000, E1  +407.021, E3 -312720.277}
SPL {X  -159.990, Y  +583.515, Z    +0.000, E1  +407.019, E3 -312729.917}
SPL {X  -159.990, Y  +589.675, Z    +0.000, E1  +407.042, E3 -312742.055}
SPL {X  -159.990, Y  +596.627, Z    +0.000, E1  +407.034, E3 -312755.795}
SPL {X  -159.990, Y  +602.039, Z    +0.000, E1  +407.021, E3 -312766.502}
SPL {X  -159.990, Y  +607.106, Z    +0.000, E1  +407.028, E3 -312776.509}
SPL {X  -159.990, Y  +612.418, Z    +0.000, E1  +407.023, E3 -312787.020}
SPL {X  -159.990, Y  +618.496, Z    +0.000, E1  +407.049, E3 -312798.987}
SPL {X  -159.990, Y  +624.357, Z    +0.000, E1  +407.020, E3 -312810.613}
SPL {X  -159.990, Y  +629.711, Z    +0.000, E1  +407.034, E3 -312821.182}
SPL {X  -159.990, Y  +635.041, Z    +0.000, E1  +407.022, E3 -312831.727}
SPL {X  -159.990, Y  +639.998, Z    +0.000, E1  +407.027, E3 -312841.519}
SPL {X  -159.990, Y  +646.188, Z    +0.000, E1  +407.041, E3 -312853.745}
SPL {X  -159.990, Y  +652.067, Z    +0.000, E1  +407.023, E3 -312865.381}
SPL {X  -159.990, Y  +657.109, Z    +0.000, E1  +407.025, E3 -312875.360}
SPL {X  -159.990, Y  +662.651, Z    +0.000, E1  +407.027, E3 -312886.316}
SPL {X  -159.990, Y  +668.015, Z    +0.000, E1  +407.025, E3 -312896.916}
SPL {X  -159.972, Y  +673.909, Z    +0.000, E1  +407.029, E3 -312908.581}
SPL {X  -159.776, Y  +679.772, Z    +0.000, E1  +406.992, E3 -312920.382}
SPL {X  -159.384, Y  +685.411, Z    +0.000, E1  +406.921, E3 -312931.944}
SPL {X  -158.839, Y  +690.657, Z    +0.000, E1  +406.819, E3 -312942.898}
SPL {X  -157.875, Y  +697.431, Z    +0.000, E1  +406.688, E3 -312957.237}
SPL {X  -156.719, Y  +703.686, Z    +0.000, E1  +406.438, E3 -312970.846}
SPL {X  -155.778, Y  +707.970, Z    +0.000, E1  +406.262, E3 -312980.321}
SPL {X  -154.419, Y  +713.351, Z    +0.000, E1  +406.025, E3 -312992.353}
SPL {X  -152.913, Y  +718.557, Z    +0.000, E1  +405.729, E3 -313004.205}
SPL {X  -151.262, Y  +723.621, Z    +0.000, E1  +405.429, E3 -313015.871}
SPL {X  -149.074, Y  +729.584, Z    +0.000, E1  +405.040, E3 -313029.800}
SPL {X  -142.577, Y  +744.086, Z    +0.000, E1  +400.686, E3 -313096.006}
ENDSPLINE

SPLINE
SPL {X  -152.566, Y  +719.671, Z    +0.000, E1  +387.682, E3 -313166.477}
SPL {X  -158.253, Y  +695.011, Z    +0.000, E1  +375.913, E3 -313183.148}
SPL {X  -159.486, Y  +684.192, Z    +0.000, E1  +369.965, E3 -313187.095}
SPL {X  -159.898, Y  +676.924, Z    +0.000, E1  +365.683, E3 -313188.793}
SPL {X  -159.990, Y  +671.720, Z    +0.000, E1  +362.298, E3 -313189.633}
SPL {X  -159.990, Y  +668.164, Z    +0.000, E1  +359.695, E3 -313190.048}
SPL {X  -159.990, Y  +665.062, Z    +0.000, E1  +356.961, E3 -313190.388}
SPL {X  -159.990, Y  +660.795, Z    +0.000, E1  +352.651, E3 -313191.051}
SPL {X  -159.990, Y  +654.574, Z    +0.000, E1  +345.673, E3 -313192.505}
SPL {X  -159.990, Y  +644.002, Z    +0.000, E1  +334.724, E3 -313196.702}
SPL {X  -159.990, Y  +611.706, Z    +0.000, E1  +317.244, E3 -313221.124}
SPL {X  -159.990, Y  +571.318, Z    +0.000, E1  +312.417, E3 -313274.508}
SPL {X  -159.990, Y  +564.395, Z    +0.000, E1  +312.373, E3 -313287.866}
SPL {X  -159.990, Y  +555.871, Z    +0.000, E1  +312.389, E3 -313304.415}
SPL {X  -159.990, Y  +549.223, Z    +0.000, E1  +312.413, E3 -313317.338}
SPL {X  -159.990, Y  +542.502, Z    +0.000, E1  +312.392, E3 -313330.335}
SPL {X  -159.990, Y  +534.538, Z    +0.000, E1  +312.385, E3 -313345.740}
SPL {X  -159.990, Y  +525.893, Z    +0.000, E1  +312.375, E3 -313362.496}
SPL {X  -159.990, Y  +516.322, Z    +0.000, E1  +312.366, E3 -313381.036}
SPL {X  -159.990, Y  +507.203, Z    +0.000, E1  +312.383, E3 -313398.739}
ENDSPLINE

SPLINE
SPL {X  -159.990, Y  +518.404, Z    +0.000, E1  +319.229, E3 -313414.837}
ENDSPLINE

SPLINE
SPL {X  -159.990, Y  +509.980, Z    +0.000, E1  +318.692, E3 -313432.240}
SPL {X  -159.990, Y  +499.983, Z    +0.000, E1  +317.561, E3 -313449.135}
SPL {X  -159.990, Y  +490.062, Z    +0.000, E1  +316.490, E3 -313465.418}
SPL {X  -159.990, Y  +479.678, Z    +0.000, E1  +315.383, E3 -313481.638}
SPL {X  -159.990, Y  +470.785, Z    +0.000, E1  +314.453, E3 -313494.871}
SPL {X  -159.990, Y  +463.371, Z    +0.000, E1  +313.690, E3 -313505.597}
SPL {X  -159.990, Y  +453.200, Z    +0.000, E1  +312.569, E3 -313519.236}
SPL {X  -159.990, Y  +441.904, Z    +0.000, E1  +311.574, E3 -313534.949}
SPL {X  -159.990, Y  +434.881, Z    +0.000, E1  +311.481, E3 -313547.498}
SPL {X  -159.990, Y  +429.614, Z    +0.000, E1  +311.486, E3 -313557.387}
SPL {X  -159.990, Y  +423.677, Z    +0.000, E1  +311.471, E3 -313568.499}
SPL {X  -159.990, Y  +417.714, Z    +0.000, E1  +311.484, E3 -313579.709}
SPL {X  -159.990, Y  +412.449, Z    +0.000, E1  +311.483, E3 -313589.569}
SPL {X  -159.990, Y  +406.256, Z    +0.000, E1  +311.459, E3 -313601.136}
SPL {X  -159.990, Y  +399.971, Z    +0.000, E1  +311.480, E3 -313612.951}
SPL {X  -159.990, Y  +394.711, Z    +0.000, E1  +311.476, E3 -313622.810}
SPL {X  -159.990, Y  +387.710, Z    +0.000, E1  +311.455, E3 -313635.933}
SPL {X  -159.984, Y  +381.116, Z    +0.000, E1  +311.484, E3 -313648.350}
SPL {X  -159.797, Y  +374.648, Z    +0.000, E1  +311.491, E3 -313660.644}
SPL {X  -159.230, Y  +366.920, Z    +0.000, E1  +311.592, E3 -313675.744}
SPL {X  -158.297, Y  +359.284, Z    +0.000, E1  +311.753, E3 -313691.044}
SPL {X  -157.042, Y  +351.926, Z    +0.000, E1  +311.986, E3 -313706.167}
SPL {X  -155.408, Y  +344.485, Z    +0.000, E1  +312.267, E3 -313721.796}
SPL {X  -153.753, Y  +338.264, Z    +0.000, E1  +312.613, E3 -313735.225}
SPL {X  -152.142, Y  +333.005, Z    +0.000, E1  +312.891, E3 -313746.699}
SPL {X  -150.309, Y  +327.691, Z    +0.000, E1  +313.264, E3 -313758.553}
SPL {X  -148.834, Y  +323.804, Z    +0.000, E1  +313.556, E3 -313767.316}
SPL {X  -147.343, Y  +320.157, Z    +0.000, E1  +313.838, E3 -313775.606}
SPL {X  -142.380, Y  +309.529, Z    +0.000, E1  +319.953, E3 -313848.367}
ENDSPLINE

SPLINE
SPL {X  -153.420, Y  +337.122, Z    +0.000, E1  +333.501, E3 -313905.865}
SPL {X  -157.288, Y  +353.220, Z    +0.000, E1  +341.134, E3 -313917.910}
SPL {X  -159.049, Y  +365.172, Z    +0.000, E1  +347.392, E3 -313923.464}
SPL {X  -159.749, Y  +373.719, Z    +0.000, E1  +352.250, E3 -313926.084}
SPL {X  -159.988, Y  +381.741, Z    +0.000, E1  +357.172, E3 -313927.559}
SPL {X  -159.990, Y  +386.092, Z    +0.000, E1  +360.442, E3 -313928.108}
SPL {X  -159.990, Y  +388.564, Z    +0.000, E1  +362.561, E3 -313928.408}
SPL {X  -159.990, Y  +392.444, Z    +0.000, E1  +366.277, E3 -313929.029}
SPL {X  -159.990, Y  +398.585, Z    +0.000, E1  +372.930, E3 -313930.409}
SPL {X  -159.990, Y  +408.423, Z    +0.000, E1  +383.302, E3 -313933.943}
SPL {X  -159.990, Y  +438.418, Z    +0.000, E1  +401.067, E3 -313955.516}
SPL {X  -159.990, Y  +482.913, Z    +0.000, E1  +407.036, E3 -314014.870}
SPL {X  -159.990, Y  +489.230, Z    +0.000, E1  +407.019, E3 -314027.382}
SPL {X  -159.990, Y  +495.241, Z    +0.000, E1  +407.026, E3 -314039.261}
SPL {X  -159.990, Y  +501.001, Z    +0.000, E1  +407.020, E3 -314050.638}
SPL {X  -159.990, Y  +506.758, Z    +0.000, E1  +407.038, E3 -314061.984}
SPL {X  -159.990, Y  +512.807, Z    +0.000, E1  +407.022, E3 -314073.975}
SPL {X  -159.990, Y  +518.043, Z    +0.000, E1  +407.016, E3 -314084.352}
SPL {X  -159.990, Y  +525.485, Z    +0.000, E1  +407.063, E3 -314098.997}
SPL {X  -159.990, Y  +533.771, Z    +0.000, E1  +407.034, E3 -314115.427}
SPL {X  -159.990, Y  +540.264, Z    +0.000, E1  +407.020, E3 -314128.283}
SPL {X  -159.990, Y  +547.787, Z    +0.000, E1  +407.067, E3 -314143.084}
SPL {X  -159.990, Y  +554.843, Z    +0.000, E1  +407.014, E3 -314157.120}
SPL {X  -159.990, Y  +560.453, Z    +0.000, E1  +407.023, E3 -314168.203}
SPL {X  -159.990, Y  +566.612, Z    +0.000, E1  +407.022, E3 -314180.385}
SPL {X  -159.990, Y  +572.901, Z    +0.000, E1  +407.028, E3 -314192.797}
SPL {X  -159.990, Y  +578.640, Z    +0.000, E1  +407.021, E3 -314204.148}
SPL {X  -159.990, Y  +583.515, Z    +0.000, E1  +407.019, E3 -314213.788}
SPL {X  -159.990, Y  +589.675, Z    +0.000, E1  +407.042, E3 -314225.926}
SPL {X  -159.990, Y  +596.627, Z    +0.000, E1  +407.034, E3 -314239.666}
SPL {X  -159.990, Y  +602.039, Z    +0.000, E1  +407.021, E3 -314250.372}
SPL {X  -159.990, Y  +607.106, Z    +0.000, E1  +407.028, E3 -314260.380}
SPL {X  -159.990, Y  +612.418, Z    +0.000, E1  +407.023, E3 -314270.891}
SPL {X  -159.990, Y  +618.496, Z    +0.000, E1  +407.049, E3 -314282.858}
SPL {X  -159.990, Y  +624.357, Z    +0.000, E1  +407.020, E3 -314294.484}
SPL {X  -159.990, Y  +629.711, Z    +0.000, E1  +407.034, E3 -314305.053}
SPL {X  -159.990, Y  +635.041, Z    +0.000, E1  +407.022, E3 -314315.598}
SPL {X  -159.990, Y  +642.261, Z    +0.000, E1  +407.074, E3 -314329.798}
SPL {X  -159.990, Y  +650.752, Z    +0.000, E1  +407.046, E3 -314346.625}
SPL {X  -159.990, Y  +657.109, Z    +0.000, E1  +407.025, E3 -314359.231}
SPL {X  -159.990, Y  +662.651, Z    +0.000, E1  +407.027, E3 -314370.187}
SPL {X  -159.990, Y  +668.015, Z    +0.000, E1  +407.025, E3 -314380.787}
SPL {X  -159.972, Y  +673.909, Z    +0.000, E1  +407.029, E3 -314392.452}
SPL {X  -159.776, Y  +679.772, Z    +0.000, E1  +406.992, E3 -314404.253}
SPL {X  -159.384, Y  +685.411, Z    +0.000, E1  +406.921, E3 -314415.815}
SPL {X  -158.839, Y  +690.657, Z    +0.000, E1  +406.819, E3 -314426.769}
SPL {X  -157.875, Y  +697.431, Z    +0.000, E1  +406.688, E3 -314441.108}
SPL {X  -156.719, Y  +703.686, Z    +0.000, E1  +406.438, E3 -314454.717}
SPL {X  -155.778, Y  +707.970, Z    +0.000, E1  +406.262, E3 -314464.192}
SPL {X  -154.419, Y  +713.351, Z    +0.000, E1  +406.025, E3 -314476.224}
SPL {X  -152.913, Y  +718.557, Z    +0.000, E1  +405.729, E3 -314488.076}
SPL {X  -151.262, Y  +723.621, Z    +0.000, E1  +405.429, E3 -314499.742}
SPL {X  -149.964, Y  +727.247, Z    +0.000, E1  +405.152, E3 -314508.246}
SPL {X  -148.611, Y  +730.759, Z    +0.000, E1  +404.909, E3 -314516.507}
SPL {X  -142.577, Y  +744.086, Z    +0.000, E1  +400.686, E3 -314579.877}
ENDSPLINE

SPLINE
SPL {X  -152.566, Y  +719.671, Z    +0.000, E1  +387.682, E3 -314650.348}
SPL {X  -158.253, Y  +695.011, Z    +0.000, E1  +375.913, E3 -314667.019}
SPL {X  -159.486, Y  +684.192, Z    +0.000, E1  +369.965, E3 -314670.966}
SPL {X  -159.898, Y  +676.924, Z    +0.000, E1  +365.683, E3 -314672.664}
SPL {X  -159.990, Y  +671.720, Z    +0.000, E1  +362.298, E3 -314673.504}
SPL {X  -159.990, Y  +668.164, Z    +0.000, E1  +359.695, E3 -314673.919}
SPL {X  -159.990, Y  +665.062, Z    +0.000, E1  +356.961, E3 -314674.259}
SPL {X  -159.990, Y  +660.795, Z    +0.000, E1  +352.651, E3 -314674.922}
SPL {X  -159.990, Y  +654.574, Z    +0.000, E1  +345.673, E3 -314676.376}
SPL {X  -159.990, Y  +647.816, Z    +0.000, E1  +338.252, E3 -314678.628}
SPL {X  -159.990, Y  +640.751, Z    +0.000, E1  +331.747, E3 -314682.221}
SPL {X  -159.990, Y  +611.706, Z    +0.000, E1  +317.244, E3 -314704.995}
SPL {X  -159.990, Y  +571.318, Z    +0.000, E1  +312.417, E3 -314758.379}
SPL {X  -159.990, Y  +564.395, Z    +0.000, E1  +312.373, E3 -314771.737}
SPL {X  -159.990, Y  +555.871, Z    +0.000, E1  +312.389, E3 -314788.285}
SPL {X  -159.990, Y  +549.223, Z    +0.000, E1  +312.413, E3 -314801.209}
SPL {X  -159.990, Y  +542.502, Z    +0.000, E1  +312.392, E3 -314814.206}
SPL {X  -159.990, Y  +536.986, Z    +0.000, E1  +312.423, E3 -314824.927}
SPL {X  -159.990, Y  +532.938, Z    +0.000, E1  +312.415, E3 -314832.753}
SPL {X  -159.990, Y  +527.222, Z    +0.000, E1  +312.401, E3 -314843.819}
SPL {X  -159.990, Y  +520.237, Z    +0.000, E1  +312.390, E3 -314857.349}
SPL {X  -159.990, Y  +514.002, Z    +0.000, E1  +312.418, E3 -314869.484}
SPL {X  -159.990, Y  +507.203, Z    +0.000, E1  +312.383, E3 -314882.610}
ENDSPLINE

SPLINE
SPL {X  -159.990, Y  +517.758, Z    +0.000, E1  +318.109, E3 -314893.183}
ENDSPLINE

SPLINE
SPL {X  -159.990, Y  +516.975, Z    +0.000, E1  +319.588, E3 -314904.246}
SPL {X  -159.990, Y  +508.583, Z    +0.000, E1  +318.552, E3 -314918.551}
SPL {X  -159.990, Y  +502.438, Z    +0.000, E1  +317.876, E3 -314929.054}
SPL {X  -159.990, Y  +494.810, Z    +0.000, E1  +316.979, E3 -314941.471}
SPL {X  -159.990, Y  +485.551, Z    +0.000, E1  +316.053, E3 -314956.659}
SPL {X  -159.990, Y  +477.585, Z    +0.000, E1  +315.156, E3 -314968.570}
SPL {X  -159.990, Y  +470.785, Z    +0.000, E1  +314.453, E3 -314978.742}
SPL {X  -159.990, Y  +463.371, Z    +0.000, E1  +313.690, E3 -314989.468}
SPL {X  -159.990, Y  +455.469, Z    +0.000, E1  +312.807, E3 -314999.994}
SPL {X  -159.990, Y  +445.848, Z    +0.000, E1  +311.866, E3 -315013.086}
SPL {X  -159.990, Y  +436.400, Z    +0.000, E1  +311.449, E3 -315028.467}
SPL {X  -159.990, Y  +429.614, Z    +0.000, E1  +311.486, E3 -315041.258}
SPL {X  -159.990, Y  +423.677, Z    +0.000, E1  +311.471, E3 -315052.370}
SPL {X  -159.990, Y  +417.714, Z    +0.000, E1  +311.484, E3 -315063.580}
SPL {X  -159.990, Y  +412.449, Z    +0.000, E1  +311.483, E3 -315073.440}
SPL {X  -159.990, Y  +406.256, Z    +0.000, E1  +311.459, E3 -315085.007}
SPL {X  -159.990, Y  +399.971, Z    +0.000, E1  +311.480, E3 -315096.822}
SPL {X  -159.990, Y  +394.711, Z    +0.000, E1  +311.476, E3 -315106.680}
SPL {X  -159.990, Y  +387.710, Z    +0.000, E1  +311.455, E3 -315119.804}
SPL {X  -159.966, Y  +379.751, Z    +0.000, E1  +311.465, E3 -315134.768}
SPL {X  -159.734, Y  +373.449, Z    +0.000, E1  +311.528, E3 -315146.872}
SPL {X  -159.358, Y  +368.299, Z    +0.000, E1  +311.595, E3 -315156.930}
SPL {X  -158.689, Y  +362.140, Z    +0.000, E1  +311.691, E3 -315169.157}
SPL {X  -157.692, Y  +355.479, Z    +0.000, E1  +311.882, E3 -315182.716}
SPL {X  -156.759, Y  +350.510, Z    +0.000, E1  +312.069, E3 -315193.032}
SPL {X  -155.408, Y  +344.485, Z    +0.000, E1  +312.267, E3 -315205.667}
SPL {X  -153.753, Y  +338.264, Z    +0.000, E1  +312.613, E3 -315219.096}
SPL {X  -152.142, Y  +333.005, Z    +0.000, E1  +312.891, E3 -315230.570}
SPL {X  -150.309, Y  +327.691, Z    +0.000, E1  +313.264, E3 -315242.424}
SPL {X  -148.834, Y  +323.804, Z    +0.000, E1  +313.556, E3 -315251.187}
SPL {X  -147.343, Y  +320.157, Z    +0.000, E1  +313.838, E3 -315259.477}
SPL {X  -142.380, Y  +309.529, Z    +0.000, E1  +319.953, E3 -315332.238}
ENDSPLINE

SPLINE
SPL {X  -153.420, Y  +337.122, Z    +0.000, E1  +333.501, E3 -315389.736}
SPL {X  -157.288, Y  +353.220, Z    +0.000, E1  +341.134, E3 -315401.781}
SPL {X  -159.049, Y  +365.172, Z    +0.000, E1  +347.392, E3 -315407.335}
SPL {X  -159.749, Y  +373.719, Z    +0.000, E1  +352.250, E3 -315409.955}
SPL {X  -159.988, Y  +381.741, Z    +0.000, E1  +357.172, E3 -315411.430}
SPL {X  -159.990, Y  +387.352, Z    +0.000, E1  +361.387, E3 -315412.132}
SPL {X  -159.990, Y  +392.444, Z    +0.000, E1  +366.277, E3 -315412.900}
SPL {X  -159.990, Y  +398.585, Z    +0.000, E1  +372.930, E3 -315414.280}
SPL {X  -159.990, Y  +408.423, Z    +0.000, E1  +383.302, E3 -315417.814}
SPL {X  -159.990, Y  +438.418, Z    +0.000, E1  +401.067, E3 -315439.387}
SPL {X  -159.990, Y  +482.913, Z    +0.000, E1  +407.036, E3 -315498.741}
SPL {X  -159.990, Y  +489.230, Z    +0.000, E1  +407.019, E3 -315511.253}
SPL {X  -159.990, Y  +495.241, Z    +0.000, E1  +407.026, E3 -315523.132}
SPL {X  -159.990, Y  +501.001, Z    +0.000, E1  +407.020, E3 -315534.509}
SPL {X  -159.990, Y  +506.758, Z    +0.000, E1  +407.038, E3 -315545.855}
SPL {X  -159.990, Y  +512.807, Z    +0.000, E1  +407.022, E3 -315557.846}
SPL {X  -159.990, Y  +518.043, Z    +0.000, E1  +407.016, E3 -315568.223}
SPL {X  -159.990, Y  +523.058, Z    +0.000, E1  +407.015, E3 -315578.139}
SPL {X  -159.990, Y  +527.746, Z    +0.000, E1  +407.012, E3 -315587.413}
SPL {X  -159.990, Y  +533.771, Z    +0.000, E1  +407.034, E3 -315599.298}
SPL {X  -159.990, Y  +542.379, Z    +0.000, E1  +407.067, E3 -315616.267}
SPL {X  -159.990, Y  +549.846, Z    +0.000, E1  +407.016, E3 -315631.113}
SPL {X  -159.990, Y  +554.843, Z    +0.000, E1  +407.014, E3 -315640.991}
SPL {X  -159.990, Y  +560.453, Z    +0.000, E1  +407.023, E3 -315652.074}
SPL {X  -159.990, Y  +566.612, Z    +0.000, E1  +407.022, E3 -315664.256}
SPL {X  -159.990, Y  +572.901, Z    +0.000, E1  +407.028, E3 -315676.668}
SPL {X  -159.990, Y  +578.640, Z    +0.000, E1  +407.021, E3 -315688.019}
SPL {X  -159.990, Y  +583.515, Z    +0.000, E1  +407.019, E3 -315697.659}
SPL {X  -159.990, Y  +589.675, Z    +0.000, E1  +407.042, E3 -315709.797}
SPL {X  -159.990, Y  +596.627, Z    +0.000, E1  +407.034, E3 -315723.537}
SPL {X  -159.990, Y  +602.039, Z    +0.000, E1  +407.021, E3 -315734.243}
SPL {X  -159.990, Y  +607.106, Z    +0.000, E1  +407.028, E3 -315744.251}
SPL {X  -159.990, Y  +612.418, Z    +0.000, E1  +407.023, E3 -315754.762}
SPL {X  -159.990, Y  +618.496, Z    +0.000, E1  +407.049, E3 -315766.729}
SPL {X  -159.990, Y  +624.357, Z    +0.000, E1  +407.020, E3 -315778.355}
SPL {X  -159.990, Y  +629.711, Z    +0.000, E1  +407.034, E3 -315788.924}
SPL {X  -159.990, Y  +635.041, Z    +0.000, E1  +407.022, E3 -315799.469}
SPL {X  -159.990, Y  +639.998, Z    +0.000, E1  +407.027, E3 -315809.261}
SPL {X  -159.990, Y  +646.188, Z    +0.000, E1  +407.041, E3 -315821.487}
SPL {X  -159.990, Y  +652.067, Z    +0.000, E1  +407.023, E3 -315833.123}
SPL {X  -159.990, Y  +657.109, Z    +0.000, E1  +407.025, E3 -315843.102}
SPL {X  -159.990, Y  +662.651, Z    +0.000, E1  +407.027, E3 -315854.058}
SPL {X  -159.990, Y  +668.015, Z    +0.000, E1  +407.025, E3 -315864.658}
SPL {X  -159.972, Y  +673.909, Z    +0.000, E1  +407.029, E3 -315876.323}
SPL {X  -159.776, Y  +679.772, Z    +0.000, E1  +406.992, E3 -315888.124}
SPL {X  -159.384, Y  +685.411, Z    +0.000, E1  +406.921, E3 -315899.685}
SPL {X  -158.839, Y  +690.657, Z    +0.000, E1  +406.819, E3 -315910.640}
SPL {X  -157.875, Y  +697.431, Z    +0.000, E1  +406.688, E3 -315924.979}
SPL {X  -156.719, Y  +703.686, Z    +0.000, E1  +406.438, E3 -315938.588}
SPL {X  -155.778, Y  +707.970, Z    +0.000, E1  +406.262, E3 -315948.063}
SPL {X  -154.419, Y  +713.351, Z    +0.000, E1  +406.025, E3 -315960.095}
SPL {X  -152.913, Y  +718.557, Z    +0.000, E1  +405.729, E3 -315971.947}
SPL {X  -151.262, Y  +723.621, Z    +0.000, E1  +405.429, E3 -315983.613}
SPL {X  -149.964, Y  +727.247, Z    +0.000, E1  +405.152, E3 -315992.117}
SPL {X  -148.611, Y  +730.759, Z    +0.000, E1  +404.909, E3 -316000.378}
SPL {X  -142.577, Y  +744.086, Z    +0.000, E1  +400.686, E3 -316063.748}
ENDSPLINE

SPLINE
SPL {X  -152.566, Y  +719.671, Z    +0.000, E1  +387.682, E3 -316134.219}
SPL {X  -158.253, Y  +695.011, Z    +0.000, E1  +375.913, E3 -316150.890}
SPL {X  -159.486, Y  +684.192, Z    +0.000, E1  +369.965, E3 -316154.837}
SPL {X  -159.898, Y  +676.924, Z    +0.000, E1  +365.683, E3 -316156.535}
SPL {X  -159.990, Y  +671.720, Z    +0.000, E1  +362.298, E3 -316157.375}
SPL {X  -159.990, Y  +668.164, Z    +0.000, E1  +359.695, E3 -316157.790}
SPL {X  -159.990, Y  +665.062, Z    +0.000, E1  +356.961, E3 -316158.130}
SPL {X  -159.990, Y  +660.795, Z    +0.000, E1  +352.651, E3 -316158.793}
SPL {X  -159.990, Y  +654.574, Z    +0.000, E1  +345.673, E3 -316160.247}
SPL {X  -159.990, Y  +647.816, Z    +0.000, E1  +338.252, E3 -316162.499}
SPL {X  -159.990, Y  +640.751, Z    +0.000, E1  +331.747, E3 -316166.092}
SPL {X  -159.990, Y  +611.706, Z    +0.000, E1  +317.244, E3 -316188.866}
SPL {X  -159.990, Y  +567.814, Z    +0.000, E1  +312.360, E3 -316248.956}
SPL {X  -159.990, Y  +557.302, Z    +0.000, E1  +312.348, E3 -316269.319}
SPL {X  -159.990, Y  +549.223, Z    +0.000, E1  +312.413, E3 -316285.080}
SPL {X  -159.990, Y  +542.502, Z    +0.000, E1  +312.392, E3 -316298.077}
SPL {X  -159.990, Y  +534.538, Z    +0.000, E1  +312.385, E3 -316313.482}
SPL {X  -159.990, Y  +525.893, Z    +0.000, E1  +312.375, E3 -316330.238}
SPL {X  -159.990, Y  +518.864, Z    +0.000, E1  +312.415, E3 -316343.920}
SPL {X  -159.990, Y  +512.328, Z    +0.000, E1  +312.388, E3 -316356.554}
SPL {X  -159.990, Y  +505.755, Z    +0.000, E1  +312.413, E3 -316369.331}
ENDSPLINE

SPLINE
SPL {X  -159.990, Y  +517.758, Z    +0.000, E1  +318.109, E3 -316377.054}
ENDSPLINE

SPLINE
SPL {X  -159.990, Y  +516.975, Z    +0.000, E1  +319.588, E3 -316388.117}
SPL {X  -159.990, Y  +508.583, Z    +0.000, E1  +318.552, E3 -316402.422}
SPL {X  -159.990, Y  +499.983, Z    +0.000, E1  +317.561, E3 -316416.877}
SPL {X  -159.990, Y  +492.624, Z    +0.000, E1  +316.776, E3 -316428.981}
SPL {X  -159.990, Y  +485.551, Z    +0.000, E1  +316.053, E3 -316440.530}
SPL {X  -159.990, Y  +477.585, Z    +0.000, E1  +315.156, E3 -316452.441}
SPL {X  -159.990, Y  +468.709, Z    +0.000, E1  +314.219, E3 -316465.619}
SPL {X  -159.990, Y  +457.446, Z    +0.000, E1  +313.017, E3 -316481.271}
SPL {X  -159.990, Y  +449.689, Z    +0.000, E1  +312.264, E3 -316491.855}
SPL {X  -159.990, Y  +441.904, Z    +0.000, E1  +311.574, E3 -316502.691}
SPL {X  -159.990, Y  +434.881, Z    +0.000, E1  +311.481, E3 -316515.240}
SPL {X  -159.990, Y  +429.614, Z    +0.000, E1  +311.486, E3 -316525.129}
SPL {X  -159.990, Y  +423.677, Z    +0.000, E1  +311.471, E3 -316536.240}
SPL {X  -159.990, Y  +417.714, Z    +0.000, E1  +311.484, E3 -316547.451}
SPL {X  -159.990, Y  +412.449, Z    +0.000, E1  +311.483, E3 -316557.311}
SPL {X  -159.990, Y  +406.256, Z    +0.000, E1  +311.459, E3 -316568.878}
SPL {X  -159.990, Y  +399.971, Z    +0.000, E1  +311.480, E3 -316580.693}
SPL {X  -159.990, Y  +392.623, Z    +0.000, E1  +311.440, E3 -316594.424}
SPL {X  -159.990, Y  +385.787, Z    +0.000, E1  +311.488, E3 -316607.331}
SPL {X  -159.966, Y  +379.751, Z    +0.000, E1  +311.465, E3 -316618.639}
SPL {X  -159.734, Y  +373.449, Z    +0.000, E1  +311.528, E3 -316630.743}
SPL {X  -159.358, Y  +368.299, Z    +0.000, E1  +311.595, E3 -316640.801}
SPL {X  -158.689, Y  +362.140, Z    +0.000, E1  +311.691, E3 -316653.028}
SPL {X  -157.958, Y  +357.080, Z    +0.000, E1  +311.860, E3 -316663.342}
SPL {X  -157.042, Y  +351.926, Z    +0.000, E1  +311.986, E3 -316673.909}
SPL {X  -155.944, Y  +346.747, Z    +0.000, E1  +312.219, E3 -316684.810}
SPL {X  -154.984, Y  +342.790, Z    +0.000, E1  +312.392, E3 -316693.224}
SPL {X  -153.753, Y  +338.264, Z    +0.000, E1  +312.613, E3 -316702.967}
SPL {X  -152.142, Y  +333.005, Z    +0.000, E1  +312.891, E3 -316714.441}
SPL {X  -150.309, Y  +327.691, Z    +0.000, E1  +313.264, E3 -316726.295}
SPL {X  -148.834, Y  +323.804, Z    +0.000, E1  +313.556, E3 -316735.058}
SPL {X  -147.343, Y  +320.157, Z    +0.000, E1  +313.838, E3 -316743.348}
SPL {X  -142.380, Y  +309.529, Z    +0.000, E1  +319.953, E3 -316816.109}
ENDSPLINE

SPLINE
SPL {X  -153.420, Y  +337.122, Z    +0.000, E1  +333.501, E3 -316873.607}
SPL {X  -157.288, Y  +353.220, Z    +0.000, E1  +341.134, E3 -316885.652}
SPL {X  -159.049, Y  +365.172, Z    +0.000, E1  +347.392, E3 -316891.205}
SPL {X  -159.749, Y  +373.719, Z    +0.000, E1  +352.250, E3 -316893.826}
SPL {X  -159.988, Y  +381.741, Z    +0.000, E1  +357.172, E3 -316895.301}
SPL {X  -159.990, Y  +386.092, Z    +0.000, E1  +360.442, E3 -316895.850}
SPL {X  -159.990, Y  +388.564, Z    +0.000, E1  +362.561, E3 -316896.150}
SPL {X  -159.990, Y  +392.444, Z    +0.000, E1  +366.277, E3 -316896.771}
SPL {X  -159.990, Y  +398.585, Z    +0.000, E1  +372.930, E3 -316898.151}
SPL {X  -159.990, Y  +408.423, Z    +0.000, E1  +383.302, E3 -316901.685}
SPL {X  -159.990, Y  +438.418, Z    +0.000, E1  +401.067, E3 -316923.258}
SPL {X  -159.990, Y  +482.913, Z    +0.000, E1  +407.036, E3 -316982.612}
SPL {X  -159.990, Y  +489.230, Z    +0.000, E1  +407.019, E3 -316995.124}
SPL {X  -159.990, Y  +495.241, Z    +0.000, E1  +407.026, E3 -317007.003}
SPL {X  -159.990, Y  +501.001, Z    +0.000, E1  +407.020, E3 -317018.380}
SPL {X  -159.990, Y  +506.758, Z    +0.000, E1  +407.038, E3 -317029.726}
SPL {X  -159.990, Y  +512.807, Z    +0.000, E1  +407.022, E3 -317041.717}
SPL {X  -159.990, Y  +518.043, Z    +0.000, E1  +407.016, E3 -317052.094}
SPL {X  -159.990, Y  +525.485, Z    +0.000, E1  +407.063, E3 -317066.739}
SPL {X  -159.990, Y  +533.771, Z    +0.000, E1  +407.034, E3 -317083.169}
SPL {X  -159.990, Y  +540.264, Z    +0.000, E1  +407.020, E3 -317096.025}
SPL {X  -159.990, Y  +547.787, Z    +0.000, E1  +407.067, E3 -317110.826}
SPL {X  -159.990, Y  +554.843, Z    +0.000, E1  +407.014, E3 -317124.862}
SPL {X  -159.990, Y  +560.453, Z    +0.000, E1  +407.023, E3 -317135.945}
SPL {X  -159.990, Y  +566.612, Z    +0.000, E1  +407.022, E3 -317148.127}
SPL {X  -159.990, Y  +572.901, Z    +0.000, E1  +407.028, E3 -317160.539}
SPL {X  -159.990, Y  +578.640, Z    +0.000, E1  +407.021, E3 -317171.890}
SPL {X  -159.990, Y  +583.515, Z    +0.000, E1  +407.019, E3 -317181.530}
SPL {X  -159.990, Y  +589.675, Z    +0.000, E1  +407.042, E3 -317193.668}
SPL {X  -159.990, Y  +596.627, Z    +0.000, E1  +407.034, E3 -317207.408}
SPL {X  -159.990, Y  +602.039, Z    +0.000, E1  +407.021, E3 -317218.114}
SPL {X  -159.990, Y  +607.106, Z    +0.000, E1  +407.028, E3 -317228.122}
SPL {X  -159.990, Y  +612.418, Z    +0.000, E1  +407.023, E3 -317238.633}
SPL {X  -159.990, Y  +618.496, Z    +0.000, E1  +407.049, E3 -317250.600}
SPL {X  -159.990, Y  +624.357, Z    +0.000, E1  +407.020, E3 -317262.226}
SPL {X  -159.990, Y  +629.711, Z    +0.000, E1  +407.034, E3 -317272.795}
SPL {X  -159.990, Y  +635.041, Z    +0.000, E1  +407.022, E3 -317283.340}
SPL {X  -159.990, Y  +642.261, Z    +0.000, E1  +407.074, E3 -317297.540}
SPL {X  -159.990, Y  +650.752, Z    +0.000, E1  +407.046, E3 -317314.367}
SPL {X  -159.990, Y  +657.109, Z    +0.000, E1  +407.025, E3 -317326.973}
SPL {X  -159.990, Y  +662.651, Z    +0.000, E1  +407.027, E3 -317337.929}
SPL {X  -159.990, Y  +668.015, Z    +0.000, E1  +407.025, E3 -317348.528}
SPL {X  -159.972, Y  +673.909, Z    +0.000, E1  +407.029, E3 -317360.194}
SPL {X  -159.776, Y  +679.772, Z    +0.000, E1  +406.992, E3 -317371.995}
SPL {X  -159.384, Y  +685.411, Z    +0.000, E1  +406.921, E3 -317383.556}
SPL {X  -158.839, Y  +690.657, Z    +0.000, E1  +406.819, E3 -317394.511}
SPL {X  -157.875, Y  +697.431, Z    +0.000, E1  +406.688, E3 -317408.850}
SPL {X  -156.719, Y  +703.686, Z    +0.000, E1  +406.438, E3 -317422.459}
SPL {X  -155.778, Y  +707.970, Z    +0.000, E1  +406.262, E3 -317431.934}
SPL {X  -154.419, Y  +713.351, Z    +0.000, E1  +406.025, E3 -317443.966}
SPL {X  -152.913, Y  +718.557, Z    +0.000, E1  +405.729, E3 -317455.818}
SPL {X  -151.262, Y  +723.621, Z    +0.000, E1  +405.429, E3 -317467.484}
SPL {X  -149.964, Y  +727.247, Z    +0.000, E1  +405.152, E3 -317475.988}
SPL {X  -148.611, Y  +730.759, Z    +0.000, E1  +404.909, E3 -317484.249}
SPL {X  -142.577, Y  +744.086, Z    +0.000, E1  +400.686, E3 -317547.619}
ENDSPLINE

SPLINE
SPL {X  -152.566, Y  +719.671, Z    +0.000, E1  +387.682, E3 -317618.090}
SPL {X  -158.253, Y  +695.011, Z    +0.000, E1  +375.913, E3 -317634.761}
SPL {X  -159.486, Y  +684.192, Z    +0.000, E1  +369.965, E3 -317638.708}
SPL {X  -159.898, Y  +676.924, Z    +0.000, E1  +365.683, E3 -317640.406}
SPL {X  -159.990, Y  +671.720, Z    +0.000, E1  +362.298, E3 -317641.246}
SPL {X  -159.990, Y  +668.164, Z    +0.000, E1  +359.695, E3 -317641.661}
SPL {X  -159.990, Y  +665.062, Z    +0.000, E1  +356.961, E3 -317642.001}
SPL {X  -159.990, Y  +660.795, Z    +0.000, E1  +352.651, E3 -317642.664}
SPL {X  -159.990, Y  +654.574, Z    +0.000, E1  +345.673, E3 -317644.118}
SPL {X  -159.990, Y  +647.816, Z    +0.000, E1  +338.252, E3 -317646.370}
SPL {X  -159.990, Y  +640.751, Z    +0.000, E1  +331.747, E3 -317649.963}
SPL {X  -159.990, Y  +611.706, Z    +0.000, E1  +317.244, E3 -317672.737}
SPL {X  -159.990, Y  +571.318, Z    +0.000, E1  +312.417, E3 -317726.121}
SPL {X  -159.990, Y  +564.395, Z    +0.000, E1  +312.373, E3 -317739.479}
SPL {X  -159.990, Y  +555.871, Z    +0.000, E1  +312.389, E3 -317756.027}
SPL {X  -159.990, Y  +549.223, Z    +0.000, E1  +312.413, E3 -317768.951}
SPL {X  -159.990, Y  +542.502, Z    +0.000, E1  +312.392, E3 -317781.948}
SPL {X  -159.990, Y  +536.986, Z    +0.000, E1  +312.423, E3 -317792.669}
SPL {X  -159.990, Y  +532.938, Z    +0.000, E1  +312.415, E3 -317800.495}
SPL {X  -159.990, Y  +527.222, Z    +0.000, E1  +312.401, E3 -317811.561}
SPL {X  -159.990, Y  +520.237, Z    +0.000, E1  +312.390, E3 -317825.091}
SPL {X  -159.990, Y  +514.002, Z    +0.000, E1  +312.418, E3 -317837.226}
SPL {X  -159.990, Y  +507.203, Z    +0.000, E1  +312.383, E3 -317850.352}
ENDSPLINE

SPLINE
SPL {X  -159.990, Y  +517.758, Z    +0.000, E1  +318.109, E3 -317860.925}
ENDSPLINE

SPLINE
SPL {X  -159.990, Y  +516.975, Z    +0.000, E1  +319.588, E3 -317871.988}
SPL {X  -159.990, Y  +508.583, Z    +0.000, E1  +318.552, E3 -317886.293}
SPL {X  -159.990, Y  +502.438, Z    +0.000, E1  +317.876, E3 -317896.796}
SPL {X  -159.990, Y  +494.810, Z    +0.000, E1  +316.979, E3 -317909.212}
SPL {X  -159.990, Y  +485.551, Z    +0.000, E1  +316.053, E3 -317924.401}
SPL {X  -159.990, Y  +477.585, Z    +0.000, E1  +315.156, E3 -317936.312}
SPL {X  -159.990, Y  +470.785, Z    +0.000, E1  +314.453, E3 -317946.484}
SPL {X  -159.990, Y  +463.371, Z    +0.000, E1  +313.690, E3 -317957.210}
SPL {X  -159.990, Y  +455.469, Z    +0.000, E1  +312.807, E3 -317967.736}
SPL {X  -159.990, Y  +445.848, Z    +0.000, E1  +311.866, E3 -317980.828}
SPL {X  -159.990, Y  +436.400, Z    +0.000, E1  +311.449, E3 -317996.209}
SPL {X  -159.990, Y  +429.614, Z    +0.000, E1  +311.486, E3 -318009.000}
SPL {X  -159.990, Y  +423.677, Z    +0.000, E1  +311.471, E3 -318020.111}
SPL {X  -159.990, Y  +417.714, Z    +0.000, E1  +311.484, E3 -318031.322}
SPL {X  -159.990, Y  +412.449, Z    +0.000, E1  +311.483, E3 -318041.182}
SPL {X  -159.990, Y  +406.256, Z    +0.000, E1  +311.459, E3 -318052.749}
SPL {X  -159.990, Y  +399.971, Z    +0.000, E1  +311.480, E3 -318064.564}
SPL {X  -159.990, Y  +394.711, Z    +0.000, E1  +311.476, E3 -318074.422}
SPL {X  -159.990, Y  +387.710, Z    +0.000, E1  +311.455, E3 -318087.546}
SPL {X  -159.966, Y  +379.751, Z    +0.000, E1  +311.465, E3 -318102.510}
SPL {X  -159.734, Y  +373.449, Z    +0.000, E1  +311.528, E3 -318114.614}
SPL {X  -159.358, Y  +368.299, Z    +0.000, E1  +311.595, E3 -318124.672}
SPL {X  -158.689, Y  +362.140, Z    +0.000, E1  +311.691, E3 -318136.899}
SPL {X  -157.692, Y  +355.479, Z    +0.000, E1  +311.882, E3 -318150.458}
SPL {X  -156.759, Y  +350.510, Z    +0.000, E1  +312.069, E3 -318160.774}
SPL {X  -155.408, Y  +344.485, Z    +0.000, E1  +312.267, E3 -318173.408}
SPL {X  -153.753, Y  +338.264, Z    +0.000, E1  +312.613, E3 -318186.838}
SPL {X  -152.142, Y  +333.005, Z    +0.000, E1  +312.891, E3 -318198.312}
SPL {X  -150.309, Y  +327.691, Z    +0.000, E1  +313.264, E3 -318210.166}
SPL {X  -148.834, Y  +323.804, Z    +0.000, E1  +313.556, E3 -318218.929}
SPL {X  -147.343, Y  +320.157, Z    +0.000, E1  +313.838, E3 -318227.219}
SPL {X  -142.380, Y  +309.529, Z    +0.000, E1  +319.953, E3 -318299.980}
ENDSPLINE

SPLINE
SPL {X  -153.420, Y  +337.122, Z    +0.000, E1  +333.501, E3 -318357.478}
SPL {X  -157.288, Y  +353.220, Z    +0.000, E1  +341.134, E3 -318369.523}
SPL {X  -159.049, Y  +365.172, Z    +0.000, E1  +347.392, E3 -318375.076}
SPL {X  -159.749, Y  +373.719, Z    +0.000, E1  +352.250, E3 -318377.697}
SPL {X  -159.988, Y  +381.741, Z    +0.000, E1  +357.172, E3 -318379.172}
SPL {X  -159.990, Y  +387.352, Z    +0.000, E1  +361.387, E3 -318379.874}
SPL {X  -159.990, Y  +392.444, Z    +0.000, E1  +366.277, E3 -318380.642}
SPL {X  -159.990, Y  +398.585, Z    +0.000, E1  +372.930, E3 -318382.022}
SPL {X  -159.990, Y  +408.423, Z    +0.000, E1  +383.302, E3 -318385.556}
SPL {X  -159.990, Y  +438.418, Z    +0.000, E1  +401.067, E3 -318407.129}
SPL {X  -159.990, Y  +482.913, Z    +0.000, E1  +407.036, E3 -318466.483}
SPL {X  -159.990, Y  +489.230, Z    +0.000, E1  +407.019, E3 -318478.995}
SPL {X  -159.990, Y  +495.241, Z    +0.000, E1  +407.026, E3 -318490.874}
SPL {X  -159.990, Y  +501.001, Z    +0.000, E1  +407.020, E3 -318502.251}
SPL {X  -159.990, Y  +506.758, Z    +0.000, E1  +407.038, E3 -318513.597}
SPL {X  -159.990, Y  +512.807, Z    +0.000, E1  +407.022, E3 -318525.588}
SPL {X  -159.990, Y  +518.043, Z    +0.000, E1  +407.016, E3 -318535.965}
SPL {X  -159.990, Y  +523.058, Z    +0.000, E1  +407.015, E3 -318545.881}
SPL {X  -159.990, Y  +527.746, Z    +0.000, E1  +407.012, E3 -318555.155}
SPL {X  -159.990, Y  +533.771, Z    +0.000, E1  +407.034, E3 -318567.040}
SPL {X  -159.990, Y  +542.379, Z    +0.000, E1  +407.067, E3 -318584.009}
SPL {X  -159.990, Y  +549.846, Z    +0.000, E1  +407.016, E3 -318598.855}
SPL {X  -159.990, Y  +554.843, Z    +0.000, E1  +407.014, E3 -318608.733}
SPL {X  -159.990, Y  +560.453, Z    +0.000, E1  +407.023, E3 -318619.816}
SPL {X  -159.990, Y  +566.612, Z    +0.000, E1  +407.022, E3 -318631.998}
SPL {X  -159.990, Y  +572.901, Z    +0.000, E1  +407.028, E3 -318644.409}
SPL {X  -159.990, Y  +578.640, Z    +0.000, E1  +407.021, E3 -318655.761}
SPL {X  -159.990, Y  +583.515, Z    +0.000, E1  +407.019, E3 -318665.401}
SPL {X  -159.990, Y  +589.675, Z    +0.000, E1  +407.042, E3 -318677.539}
SPL {X  -159.990, Y  +596.627, Z    +0.000, E1  +407.034, E3 -318691.279}
SPL {X  -159.990, Y  +602.039, Z    +0.000, E1  +407.021, E3 -318701.985}
SPL {X  -159.990, Y  +607.106, Z    +0.000, E1  +407.028, E3 -318711.993}
SPL {X  -159.990, Y  +612.418, Z    +0.000, E1  +407.023, E3 -318722.504}
SPL {X  -159.990, Y  +618.496, Z    +0.000, E1  +407.049, E3 -318734.471}
SPL {X  -159.990, Y  +624.357, Z    +0.000, E1  +407.020, E3 -318746.097}
SPL {X  -159.990, Y  +629.711, Z    +0.000, E1  +407.034, E3 -318756.666}
SPL {X  -159.990, Y  +635.041, Z    +0.000, E1  +407.022, E3 -318767.210}
SPL {X  -159.990, Y  +639.998, Z    +0.000, E1  +407.027, E3 -318777.003}
SPL {X  -159.990, Y  +646.188, Z    +0.000, E1  +407.041, E3 -318789.229}
SPL {X  -159.990, Y  +652.067, Z    +0.000, E1  +407.023, E3 -318800.865}
SPL {X  -159.990, Y  +657.109, Z    +0.000, E1  +407.025, E3 -318810.844}
SPL {X  -159.990, Y  +662.651, Z    +0.000, E1  +407.027, E3 -318821.800}
SPL {X  -159.990, Y  +668.015, Z    +0.000, E1  +407.025, E3 -318832.399}
SPL {X  -159.972, Y  +673.909, Z    +0.000, E1  +407.029, E3 -318844.065}
SPL {X  -159.776, Y  +679.772, Z    +0.000, E1  +406.992, E3 -318855.866}
SPL {X  -159.384, Y  +685.411, Z    +0.000, E1  +406.921, E3 -318867.427}
SPL {X  -158.839, Y  +690.657, Z    +0.000, E1  +406.819, E3 -318878.382}
SPL {X  -157.875, Y  +697.431, Z    +0.000, E1  +406.688, E3 -318892.721}
SPL {X  -156.719, Y  +703.686, Z    +0.000, E1  +406.438, E3 -318906.330}
SPL {X  -155.778, Y  +707.970, Z    +0.000, E1  +406.262, E3 -318915.805}
SPL {X  -154.419, Y  +713.351, Z    +0.000, E1  +406.025, E3 -318927.837}
SPL {X  -152.913, Y  +718.557, Z    +0.000, E1  +405.729, E3 -318939.689}
SPL {X  -151.262, Y  +723.621, Z    +0.000, E1  +405.429, E3 -318951.355}
SPL {X  -149.964, Y  +727.247, Z    +0.000, E1  +405.152, E3 -318959.859}
SPL {X  -148.611, Y  +730.759, Z    +0.000, E1  +404.909, E3 -318968.120}
SPL {X  -142.577, Y  +744.086, Z    +0.000, E1  +400.686, E3 -319031.490}
ENDSPLINE

SPLINE
SPL {X  -152.566, Y  +719.671, Z    +0.000, E1  +387.682, E3 -319101.960}
SPL {X  -158.253, Y  +695.011, Z    +0.000, E1  +375.913, E3 -319118.632}
SPL {X  -159.486, Y  +684.192, Z    +0.000, E1  +369.965, E3 -319122.579}
SPL {X  -159.898, Y  +676.924, Z    +0.000, E1  +365.683, E3 -319124.277}
SPL {X  -159.990, Y  +671.720, Z    +0.000, E1  +362.298, E3 -319125.117}
SPL {X  -159.990, Y  +668.164, Z    +0.000, E1  +359.695, E3 -319125.532}
SPL {X  -159.990, Y  +665.062, Z    +0.000, E1  +356.961, E3 -319125.872}
SPL {X  -159.990, Y  +660.795, Z    +0.000, E1  +352.651, E3 -319126.535}
SPL {X  -159.990, Y  +654.574, Z    +0.000, E1  +345.673, E3 -319127.989}
SPL {X  -159.990, Y  +647.816, Z    +0.000, E1  +338.252, E3 -319130.241}
SPL {X  -159.990, Y  +640.751, Z    +0.000, E1  +331.747, E3 -319133.834}
SPL {X  -159.990, Y  +611.706, Z    +0.000, E1  +317.244, E3 -319156.608}
SPL {X  -159.990, Y  +571.318, Z    +0.000, E1  +312.417, E3 -319209.992}
SPL {X  -159.990, Y  +564.395, Z    +0.000, E1  +312.373, E3 -319223.350}
SPL {X  -159.990, Y  +555.871, Z    +0.000, E1  +312.389, E3 -319239.898}
SPL {X  -159.990, Y  +549.223, Z    +0.000, E1  +312.413, E3 -319252.822}
SPL {X  -159.990, Y  +542.502, Z    +0.000, E1  +312.392, E3 -319265.819}
SPL {X  -159.990, Y  +536.986, Z    +0.000, E1  +312.423, E3 -319276.540}
SPL {X  -159.990, Y  +532.938, Z    +0.000, E1  +312.415, E3 -319284.366}
SPL {X  -159.990, Y  +527.222, Z    +0.000, E1  +312.401, E3 -319295.432}
SPL {X  -159.990, Y  +520.237, Z    +0.000, E1  +312.390, E3 -319308.962}
SPL {X  -159.990, Y  +514.002, Z    +0.000, E1  +312.418, E3 -319321.097}
SPL {X  -159.990, Y  +507.203, Z    +0.000, E1  +312.383, E3 -319334.223}
ENDSPLINE

SPLINE
SPL {X  -159.990, Y  +517.758, Z    +0.000, E1  +318.109, E3 -319344.796}
ENDSPLINE

SPLINE
SPL {X  -159.990, Y  +516.975, Z    +0.000, E1  +319.588, E3 -319355.859}
SPL {X  -159.990, Y  +508.583, Z    +0.000, E1  +318.552, E3 -319370.164}
SPL {X  -159.990, Y  +502.438, Z    +0.000, E1  +317.876, E3 -319380.667}
SPL {X  -159.990, Y  +494.810, Z    +0.000, E1  +316.979, E3 -319393.083}
SPL {X  -159.990, Y  +485.551, Z    +0.000, E1  +316.053, E3 -319408.272}
SPL {X  -159.990, Y  +477.585, Z    +0.000, E1  +315.156, E3 -319420.183}
SPL {X  -159.990, Y  +470.785, Z    +0.000, E1  +314.453, E3 -319430.355}
SPL {X  -159.990, Y  +463.371, Z    +0.000, E1  +313.690, E3 -319441.081}
SPL {X  -159.990, Y  +455.469, Z    +0.000, E1  +312.807, E3 -319451.607}
SPL {X  -159.990, Y  +445.848, Z    +0.000, E1  +311.866, E3 -319464.699}
SPL {X  -159.990, Y  +436.400, Z    +0.000, E1  +311.449, E3 -319480.080}
SPL {X  -159.990, Y  +429.614, Z    +0.000, E1  +311.486, E3 -319492.871}
SPL {X  -159.990, Y  +423.677, Z    +0.000, E1  +311.471, E3 -319503.982}
SPL {X  -159.990, Y  +417.714, Z    +0.000, E1  +311.484, E3 -319515.193}
SPL {X  -159.990, Y  +412.449, Z    +0.000, E1  +311.483, E3 -319525.053}
SPL {X  -159.990, Y  +406.256, Z    +0.000, E1  +311.459, E3 -319536.620}
SPL {X  -159.990, Y  +399.971, Z    +0.000, E1  +311.480, E3 -319548.435}
SPL {X  -159.990, Y  +392.623, Z    +0.000, E1  +311.440, E3 -319562.166}
SPL {X  -159.990, Y  +385.787, Z    +0.000, E1  +311.488, E3 -319575.073}
SPL {X  -159.966, Y  +379.751, Z    +0.000, E1  +311.465, E3 -319586.380}
SPL {X  -159.734, Y  +373.449, Z    +0.000, E1  +311.528, E3 -319598.485}
SPL {X  -159.230, Y  +366.920, Z    +0.000, E1  +311.592, E3 -319611.228}
SPL {X  -158.532, Y  +360.951, Z    +0.000, E1  +311.745, E3 -319623.202}
SPL {X  -157.692, Y  +355.479, Z    +0.000, E1  +311.882, E3 -319634.329}
SPL {X  -156.349, Y  +348.560, Z    +0.000, E1  +312.101, E3 -319648.669}
SPL {X  -154.984, Y  +342.790, Z    +0.000, E1  +312.392, E3 -319660.966}
SPL {X  -153.247, Y  +336.540, Z    +0.000, E1  +312.660, E3 -319674.401}
SPL {X  -150.765, Y  +328.959, Z    +0.000, E1  +313.136, E3 -319691.148}
SPL {X  -148.834, Y  +323.804, Z    +0.000, E1  +313.556, E3 -319702.800}
SPL {X  -147.343, Y  +320.157, Z    +0.000, E1  +313.838, E3 -319711.090}
SPL {X  -142.380, Y  +309.529, Z    +0.000, E1  +319.953, E3 -319783.851}
ENDSPLINE

SPLINE
SPL {X  -153.420, Y  +337.122, Z    +0.000, E1  +333.501, E3 -319841.349}
SPL {X  -157.288, Y  +353.220, Z    +0.000, E1  +341.134, E3 -319853.394}
SPL {X  -159.049, Y  +365.172, Z    +0.000, E1  +347.392, E3 -319858.947}
SPL {X  -159.749, Y  +373.719, Z    +0.000, E1  +352.250, E3 -319861.568}
SPL {X  -159.988, Y  +381.741, Z    +0.000, E1  +357.172, E3 -319863.043}
SPL {X  -159.990, Y  +387.352, Z    +0.000, E1  +361.387, E3 -319863.745}
SPL {X  -159.990, Y  +391.188, Z    +0.000, E1  +365.082, E3 -319864.285}
SPL {X  -159.990, Y  +395.106, Z    +0.000, E1  +369.154, E3 -319865.026}
SPL {X  -159.990, Y  +400.303, Z    +0.000, E1  +374.927, E3 -319866.348}
SPL {X  -159.990, Y  +408.423, Z    +0.000, E1  +383.302, E3 -319869.427}
SPL {X  -159.990, Y  +438.418, Z    +0.000, E1  +401.067, E3 -319891.000}
SPL {X  -159.990, Y  +482.913, Z    +0.000, E1  +407.036, E3 -319950.354}
SPL {X  -159.990, Y  +489.230, Z    +0.000, E1  +407.019, E3 -319962.866}
SPL {X  -159.990, Y  +495.241, Z    +0.000, E1  +407.026, E3 -319974.745}
SPL {X  -159.990, Y  +501.001, Z    +0.000, E1  +407.020, E3 -319986.122}
SPL {X  -159.990, Y  +506.758, Z    +0.000, E1  +407.038, E3 -319997.468}
SPL {X  -159.990, Y  +512.807, Z    +0.000, E1  +407.022, E3 -320009.459}
SPL {X  -159.990, Y  +518.043, Z    +0.000, E1  +407.016, E3 -320019.836}
SPL {X  -159.990, Y  +523.058, Z    +0.000, E1  +407.015, E3 -320029.752}
SPL {X  -159.990, Y  +527.746, Z    +0.000, E1  +407.012, E3 -320039.026}
SPL {X  -159.990, Y  +533.771, Z    +0.000, E1  +407.034, E3 -320050.911}
SPL {X  -159.990, Y  +542.379, Z    +0.000, E1  +407.067, E3 -320067.880}
SPL {X  -159.990, Y  +549.846, Z    +0.000, E1  +407.016, E3 -320082.726}
SPL {X  -159.990, Y  +554.843, Z    +0.000, E1  +407.014, E3 -320092.604}
SPL {X  -159.990, Y  +560.453, Z    +0.000, E1  +407.023, E3 -320103.687}
SPL {X  -159.990, Y  +566.612, Z    +0.000, E1  +407.022, E3 -320115.869}
SPL {X  -159.990, Y  +572.901, Z    +0.000, E1  +407.028, E3 -320128.280}
SPL {X  -159.990, Y  +578.640, Z    +0.000, E1  +407.021, E3 -320139.632}
SPL {X  -159.990, Y  +583.515, Z    +0.000, E1  +407.019, E3 -320149.272}
SPL {X  -159.990, Y  +589.675, Z    +0.000, E1  +407.042, E3 -320161.410}
SPL {X  -159.990, Y  +596.627, Z    +0.000, E1  +407.034, E3 -320175.150}
SPL {X  -159.990, Y  +602.039, Z    +0.000, E1  +407.021, E3 -320185.856}
SPL {X  -159.990, Y  +607.106, Z    +0.000, E1  +407.028, E3 -320195.864}
SPL {X  -159.990, Y  +612.418, Z    +0.000, E1  +407.023, E3 -320206.375}
SPL {X  -159.990, Y  +618.496, Z    +0.000, E1  +407.049, E3 -320218.342}
SPL {X  -159.990, Y  +624.357, Z    +0.000, E1  +407.020, E3 -320229.968}
SPL {X  -159.990, Y  +629.711, Z    +0.000, E1  +407.034, E3 -320240.537}
SPL {X  -159.990, Y  +635.041, Z    +0.000, E1  +407.022, E3 -320251.081}
SPL {X  -159.990, Y  +639.998, Z    +0.000, E1  +407.027, E3 -320260.874}
SPL {X  -159.990, Y  +646.188, Z    +0.000, E1  +407.041, E3 -320273.100}
SPL {X  -159.990, Y  +652.067, Z    +0.000, E1  +407.023, E3 -320284.736}
SPL {X  -159.990, Y  +657.109, Z    +0.000, E1  +407.025, E3 -320294.715}
SPL {X  -159.990, Y  +662.651, Z    +0.000, E1  +407.027, E3 -320305.670}
SPL {X  -159.990, Y  +668.015, Z    +0.000, E1  +407.025, E3 -320316.270}
SPL {X  -159.972, Y  +673.909, Z    +0.000, E1  +407.029, E3 -320327.936}
SPL {X  -159.776, Y  +679.772, Z    +0.000, E1  +406.992, E3 -320339.737}
SPL {X  -159.384, Y  +685.411, Z    +0.000, E1  +406.921, E3 -320351.298}
SPL {X  -158.839, Y  +690.657, Z    +0.000, E1  +406.819, E3 -320362.253}
SPL {X  -157.875, Y  +697.431, Z    +0.000, E1  +406.688, E3 -320376.592}
SPL {X  -156.719, Y  +703.686, Z    +0.000, E1  +406.438, E3 -320390.201}
SPL {X  -155.778, Y  +707.970, Z    +0.000, E1  +406.262, E3 -320399.676}
SPL {X  -154.419, Y  +713.351, Z    +0.000, E1  +406.025, E3 -320411.708}
SPL {X  -152.913, Y  +718.557, Z    +0.000, E1  +405.729, E3 -320423.559}
SPL {X  -151.262, Y  +723.621, Z    +0.000, E1  +405.429, E3 -320435.226}
SPL {X  -149.964, Y  +727.247, Z    +0.000, E1  +405.152, E3 -320443.730}
SPL {X  -148.611, Y  +730.759, Z    +0.000, E1  +404.909, E3 -320451.991}
SPL {X  -142.577, Y  +744.086, Z    +0.000, E1  +400.686, E3 -320515.361}
ENDSPLINE

SPLINE
SPL {X  -152.566, Y  +719.671, Z    +0.000, E1  +387.682, E3 -320585.831}
SPL {X  -158.253, Y  +695.011, Z    +0.000, E1  +375.913, E3 -320602.503}
SPL {X  -159.486, Y  +684.192, Z    +0.000, E1  +369.965, E3 -320606.450}
SPL {X  -159.898, Y  +676.924, Z    +0.000, E1  +365.683, E3 -320608.148}
SPL {X  -159.990, Y  +671.720, Z    +0.000, E1  +362.298, E3 -320608.988}
SPL {X  -159.990, Y  +668.164, Z    +0.000, E1  +359.695, E3 -320609.403}
SPL {X  -159.990, Y  +665.062, Z    +0.000, E1  +356.961, E3 -320609.743}
SPL {X  -159.990, Y  +660.795, Z    +0.000, E1  +352.651, E3 -320610.405}
SPL {X  -159.990, Y  +654.574, Z    +0.000, E1  +345.673, E3 -320611.860}
SPL {X  -159.990, Y  +647.816, Z    +0.000, E1  +338.252, E3 -320614.112}
SPL {X  -159.990, Y  +640.751, Z    +0.000, E1  +331.747, E3 -320617.705}
SPL {X  -159.990, Y  +611.706, Z    +0.000, E1  +317.244, E3 -320640.479}
SPL {X  -159.990, Y  +571.318, Z    +0.000, E1  +312.417, E3 -320693.863}
SPL {X  -159.990, Y  +564.395, Z    +0.000, E1  +312.373, E3 -320707.221}
SPL {X  -159.990, Y  +555.871, Z    +0.000, E1  +312.389, E3 -320723.769}
SPL {X  -159.990, Y  +549.223, Z    +0.000, E1  +312.413, E3 -320736.693}
SPL {X  -159.990, Y  +542.502, Z    +0.000, E1  +312.392, E3 -320749.690}
SPL {X  -159.990, Y  +536.986, Z    +0.000, E1  +312.423, E3 -320760.411}
SPL {X  -159.990, Y  +532.938, Z    +0.000, E1  +312.415, E3 -320768.237}
SPL {X  -159.990, Y  +527.222, Z    +0.000, E1  +312.401, E3 -320779.303}
SPL {X  -159.990, Y  +520.237, Z    +0.000, E1  +312.390, E3 -320792.833}
SPL {X  -159.990, Y  +514.002, Z    +0.000, E1  +312.418, E3 -320804.968}
SPL {X  -159.990, Y  +507.203, Z    +0.000, E1  +312.383, E3 -320818.094}
ENDSPLINE

SPLINE
SPL {X  -159.990, Y  +517.758, Z    +0.000, E1  +318.109, E3 -320828.667}
ENDSPLINE

SPLINE
SPL {X  -159.990, Y  +516.975, Z    +0.000, E1  +319.588, E3 -320839.730}
SPL {X  -159.990, Y  +508.583, Z    +0.000, E1  +318.552, E3 -320854.035}
SPL {X  -159.990, Y  +502.438, Z    +0.000, E1  +317.876, E3 -320864.538}
SPL {X  -159.990, Y  +494.810, Z    +0.000, E1  +316.979, E3 -320876.954}
SPL {X  -159.990, Y  +485.551, Z    +0.000, E1  +316.053, E3 -320892.143}
SPL {X  -159.990, Y  +477.585, Z    +0.000, E1  +315.156, E3 -320904.054}
SPL {X  -159.990, Y  +470.785, Z    +0.000, E1  +314.453, E3 -320914.226}
SPL {X  -159.990, Y  +463.371, Z    +0.000, E1  +313.690, E3 -320924.952}
SPL {X  -159.990, Y  +455.469, Z    +0.000, E1  +312.807, E3 -320935.478}
SPL {X  -159.990, Y  +445.848, Z    +0.000, E1  +311.866, E3 -320948.570}
SPL {X  -159.990, Y  +436.400, Z    +0.000, E1  +311.449, E3 -320963.951}
SPL {X  -159.990, Y  +429.614, Z    +0.000, E1  +311.486, E3 -320976.742}
SPL {X  -159.990, Y  +423.677, Z    +0.000, E1  +311.471, E3 -320987.853}
SPL {X  -159.990, Y  +417.714, Z    +0.000, E1  +311.484, E3 -320999.064}
SPL {X  -159.990, Y  +412.449, Z    +0.000, E1  +311.483, E3 -321008.924}
SPL {X  -159.990, Y  +406.256, Z    +0.000, E1  +311.459, E3 -321020.491}
SPL {X  -159.990, Y  +399.971, Z    +0.000, E1  +311.480, E3 -321032.306}
SPL {X  -159.990, Y  +394.711, Z    +0.000, E1  +311.476, E3 -321042.164}
SPL {X  -159.990, Y  +387.710, Z    +0.000, E1  +311.455, E3 -321055.287}
SPL {X  -159.966, Y  +379.751, Z    +0.000, E1  +311.465, E3 -321070.251}
SPL {X  -159.734, Y  +373.449, Z    +0.000, E1  +311.528, E3 -321082.356}
SPL {X  -159.358, Y  +368.299, Z    +0.000, E1  +311.595, E3 -321092.414}
SPL {X  -158.689, Y  +362.140, Z    +0.000, E1  +311.691, E3 -321104.641}
SPL {X  -157.692, Y  +355.479, Z    +0.000, E1  +311.882, E3 -321118.200}
SPL {X  -156.759, Y  +350.510, Z    +0.000, E1  +312.069, E3 -321128.516}
SPL {X  -155.408, Y  +344.485, Z    +0.000, E1  +312.267, E3 -321141.150}
SPL {X  -153.753, Y  +338.264, Z    +0.000, E1  +312.613, E3 -321154.580}
SPL {X  -152.142, Y  +333.005, Z    +0.000, E1  +312.891, E3 -321166.054}
SPL {X  -150.309, Y  +327.691, Z    +0.000, E1  +313.264, E3 -321177.908}
SPL {X  -148.834, Y  +323.804, Z    +0.000, E1  +313.556, E3 -321186.671}
SPL {X  -147.343, Y  +320.157, Z    +0.000, E1  +313.838, E3 -321194.961}
SPL {X  -142.380, Y  +309.529, Z    +0.000, E1  +319.953, E3 -321267.722}
ENDSPLINE

SPLINE
SPL {X  -153.420, Y  +337.122, Z    +0.000, E1  +333.501, E3 -321325.220}
SPL {X  -157.288, Y  +353.220, Z    +0.000, E1  +341.134, E3 -321337.265}
SPL {X  -159.049, Y  +365.172, Z    +0.000, E1  +347.392, E3 -321342.818}
SPL {X  -159.749, Y  +373.719, Z    +0.000, E1  +352.250, E3 -321345.439}
SPL {X  -159.988, Y  +381.741, Z    +0.000, E1  +357.172, E3 -321346.914}
SPL {X  -159.990, Y  +387.352, Z    +0.000, E1  +361.387, E3 -321347.616}
SPL {X  -159.990, Y  +392.444, Z    +0.000, E1  +366.277, E3 -321348.384}
SPL {X  -159.990, Y  +398.585, Z    +0.000, E1  +372.930, E3 -321349.764}
SPL {X  -159.990, Y  +408.423, Z    +0.000, E1  +383.302, E3 -321353.298}
SPL {X  -159.990, Y  +438.418, Z    +0.000, E1  +401.067, E3 -321374.871}
SPL {X  -159.990, Y  +482.913, Z    +0.000, E1  +407.036, E3 -321434.225}
SPL {X  -159.990, Y  +489.230, Z    +0.000, E1  +407.019, E3 -321446.737}
SPL {X  -159.990, Y  +495.241, Z    +0.000, E1  +407.026, E3 -321458.616}
SPL {X  -159.990, Y  +501.001, Z    +0.000, E1  +407.020, E3 -321469.993}
SPL {X  -159.990, Y  +506.758, Z    +0.000, E1  +407.038, E3 -321481.339}
SPL {X  -159.990, Y  +512.807, Z    +0.000, E1  +407.022, E3 -321493.330}
SPL {X  -159.990, Y  +518.043, Z    +0.000, E1  +407.016, E3 -321503.707}
SPL {X  -159.990, Y  +523.058, Z    +0.000, E1  +407.015, E3 -321513.623}
SPL {X  -159.990, Y  +527.746, Z    +0.000, E1  +407.012, E3 -321522.897}
SPL {X  -159.990, Y  +533.771, Z    +0.000, E1  +407.034, E3 -321534.782}
SPL {X  -159.990, Y  +542.379, Z    +0.000, E1  +407.067, E3 -321551.751}
SPL {X  -159.990, Y  +549.846, Z    +0.000, E1  +407.016, E3 -321566.597}
SPL {X  -159.990, Y  +554.843, Z    +0.000, E1  +407.014, E3 -321576.475}
SPL {X  -159.990, Y  +560.453, Z    +0.000, E1  +407.023, E3 -321587.558}
SPL {X  -159.990, Y  +566.612, Z    +0.000, E1  +407.022, E3 -321599.740}
SPL {X  -159.990, Y  +572.901, Z    +0.000, E1  +407.028, E3 -321612.151}
SPL {X  -159.990, Y  +578.640, Z    +0.000, E1  +407.021, E3 -321623.503}
SPL {X  -159.990, Y  +583.515, Z    +0.000, E1  +407.019, E3 -321633.143}
SPL {X  -159.990, Y  +589.675, Z    +0.000, E1  +407.042, E3 -321645.281}
SPL {X  -159.990, Y  +596.627, Z    +0.000, E1  +407.034, E3 -321659.021}
SPL {X  -159.990, Y  +602.039, Z    +0.000, E1  +407.021, E3 -321669.727}
SPL {X  -159.990, Y  +607.106, Z    +0.000, E1  +407.028, E3 -321679.735}
SPL {X  -159.990, Y  +612.418, Z    +0.000, E1  +407.023, E3 -321690.246}
SPL {X  -159.990, Y  +618.496, Z    +0.000, E1  +407.049, E3 -321702.213}
SPL {X  -159.990, Y  +624.357, Z    +0.000, E1  +407.020, E3 -321713.839}
SPL {X  -159.990, Y  +629.711, Z    +0.000, E1  +407.034, E3 -321724.408}
SPL {X  -159.990, Y  +635.041, Z    +0.000, E1  +407.022, E3 -321734.952}
SPL {X  -159.990, Y  +639.998, Z    +0.000, E1  +407.027, E3 -321744.745}
SPL {X  -159.990, Y  +646.188, Z    +0.000, E1  +407.041, E3 -321756.971}
SPL {X  -159.990, Y  +652.067, Z    +0.000, E1  +407.023, E3 -321768.607}
SPL {X  -159.990, Y  +657.109, Z    +0.000, E1  +407.025, E3 -321778.585}
SPL {X  -159.990, Y  +662.651, Z    +0.000, E1  +407.027, E3 -321789.541}
SPL {X  -159.990, Y  +668.015, Z    +0.000, E1  +407.025, E3 -321800.141}
SPL {X  -159.972, Y  +673.909, Z    +0.000, E1  +407.029, E3 -321811.807}
SPL {X  -159.776, Y  +679.772, Z    +0.000, E1  +406.992, E3 -321823.608}
SPL {X  -159.384, Y  +685.411, Z    +0.000, E1  +406.921, E3 -321835.169}
SPL {X  -158.839, Y  +690.657, Z    +0.000, E1  +406.819, E3 -321846.124}
SPL {X  -157.875, Y  +697.431, Z    +0.000, E1  +406.688, E3 -321860.463}
SPL {X  -156.719, Y  +703.686, Z    +0.000, E1  +406.438, E3 -321874.072}
SPL {X  -155.778, Y  +707.970, Z    +0.000, E1  +406.262, E3 -321883.547}
SPL {X  -154.419, Y  +713.351, Z    +0.000, E1  +406.025, E3 -321895.579}
SPL {X  -152.913, Y  +718.557, Z    +0.000, E1  +405.729, E3 -321907.430}
SPL {X  -151.262, Y  +723.621, Z    +0.000, E1  +405.429, E3 -321919.097}
SPL {X  -149.964, Y  +727.247, Z    +0.000, E1  +405.152, E3 -321927.601}
SPL {X  -148.611, Y  +730.759, Z    +0.000, E1  +404.909, E3 -321935.862}
SPL {X  -142.577, Y  +744.086, Z    +0.000, E1  +400.686, E3 -321999.232}
ENDSPLINE

SPLINE
SPL {X  -152.566, Y  +719.671, Z    +0.000, E1  +387.682, E3 -322069.702}
SPL {X  -158.253, Y  +695.011, Z    +0.000, E1  +375.913, E3 -322086.374}
SPL {X  -159.486, Y  +684.192, Z    +0.000, E1  +369.965, E3 -322090.321}
SPL {X  -159.898, Y  +676.924, Z    +0.000, E1  +365.683, E3 -322092.019}
SPL {X  -159.990, Y  +671.720, Z    +0.000, E1  +362.298, E3 -322092.859}
SPL {X  -159.990, Y  +668.164, Z    +0.000, E1  +359.695, E3 -322093.274}
SPL {X  -159.990, Y  +665.062, Z    +0.000, E1  +356.961, E3 -322093.614}
SPL {X  -159.990, Y  +660.795, Z    +0.000, E1  +352.651, E3 -322094.276}
SPL {X  -159.990, Y  +654.574, Z    +0.000, E1  +345.673, E3 -322095.731}
SPL {X  -159.990, Y  +647.816, Z    +0.000, E1  +338.252, E3 -322097.983}
SPL {X  -159.990, Y  +640.751, Z    +0.000, E1  +331.747, E3 -322101.576}
SPL {X  -159.990, Y  +611.706, Z    +0.000, E1  +317.244, E3 -322124.350}
SPL {X  -159.990, Y  +571.318, Z    +0.000, E1  +312.417, E3 -322177.734}
SPL {X  -159.990, Y  +564.395, Z    +0.000, E1  +312.373, E3 -322191.092}
SPL {X  -159.990, Y  +555.871, Z    +0.000, E1  +312.389, E3 -322207.640}
SPL {X  -159.990, Y  +549.223, Z    +0.000, E1  +312.413, E3 -322220.563}
SPL {X  -159.990, Y  +542.502, Z    +0.000, E1  +312.392, E3 -322233.561}
SPL {X  -159.990, Y  +536.986, Z    +0.000, E1  +312.423, E3 -322244.281}
SPL {X  -159.990, Y  +532.938, Z    +0.000, E1  +312.415, E3 -322252.108}
SPL {X  -159.990, Y  +527.222, Z    +0.000, E1  +312.401, E3 -322263.174}
SPL {X  -159.990, Y  +520.237, Z    +0.000, E1  +312.390, E3 -322276.704}
SPL {X  -159.990, Y  +514.002, Z    +0.000, E1  +312.418, E3 -322288.839}
SPL {X  -159.990, Y  +507.203, Z    +0.000, E1  +312.383, E3 -322301.965}
ENDSPLINE

SPLINE
SPL {X  -159.990, Y  +517.758, Z    +0.000, E1  +318.109, E3 -322312.538}
ENDSPLINE

SPLINE
SPL {X  -159.990, Y  +516.975, Z    +0.000, E1  +319.588, E3 -322323.601}
SPL {X  -159.990, Y  +508.583, Z    +0.000, E1  +318.552, E3 -322337.906}
SPL {X  -159.990, Y  +502.438, Z    +0.000, E1  +317.876, E3 -322348.409}
SPL {X  -159.990, Y  +494.810, Z    +0.000, E1  +316.979, E3 -322360.825}
SPL {X  -159.990, Y  +485.551, Z    +0.000, E1  +316.053, E3 -322376.014}
SPL {X  -159.990, Y  +477.585, Z    +0.000, E1  +315.156, E3 -322387.925}
SPL {X  -159.990, Y  +470.785, Z    +0.000, E1  +314.453, E3 -322398.097}
SPL {X  -159.990, Y  +463.371, Z    +0.000, E1  +313.690, E3 -322408.823}
SPL {X  -159.990, Y  +455.469, Z    +0.000, E1  +312.807, E3 -322419.348}
SPL {X  -159.990, Y  +445.848, Z    +0.000, E1  +311.866, E3 -322432.441}
SPL {X  -159.990, Y  +436.400, Z    +0.000, E1  +311.449, E3 -322447.822}
SPL {X  -159.990, Y  +429.614, Z    +0.000, E1  +311.486, E3 -322460.613}
SPL {X  -159.990, Y  +423.677, Z    +0.000, E1  +311.471, E3 -322471.724}
SPL {X  -159.990, Y  +417.714, Z    +0.000, E1  +311.484, E3 -322482.935}
SPL {X  -159.990, Y  +412.449, Z    +0.000, E1  +311.483, E3 -322492.795}
SPL {X  -159.990, Y  +406.256, Z    +0.000, E1  +311.459, E3 -322504.362}
SPL {X  -159.990, Y  +399.971, Z    +0.000, E1  +311.480, E3 -322516.177}
SPL {X  -159.990, Y  +392.623, Z    +0.000, E1  +311.440, E3 -322529.908}
SPL {X  -159.990, Y  +385.787, Z    +0.000, E1  +311.488, E3 -322542.815}
SPL {X  -159.966, Y  +379.751, Z    +0.000, E1  +311.465, E3 -322554.122}
SPL {X  -159.734, Y  +373.449, Z    +0.000, E1  +311.528, E3 -322566.227}
SPL {X  -159.230, Y  +366.920, Z    +0.000, E1  +311.592, E3 -322578.970}
SPL {X  -158.532, Y  +360.951, Z    +0.000, E1  +311.745, E3 -322590.944}
SPL {X  -157.692, Y  +355.479, Z    +0.000, E1  +311.882, E3 -322602.071}
SPL {X  -156.349, Y  +348.560, Z    +0.000, E1  +312.101, E3 -322616.411}
SPL {X  -154.984, Y  +342.790, Z    +0.000, E1  +312.392, E3 -322628.708}
SPL {X  -153.247, Y  +336.540, Z    +0.000, E1  +312.660, E3 -322642.143}
SPL {X  -150.765, Y  +328.959, Z    +0.000, E1  +313.136, E3 -322658.890}
SPL {X  -148.834, Y  +323.804, Z    +0.000, E1  +313.556, E3 -322670.542}
SPL {X  -147.343, Y  +320.157, Z    +0.000, E1  +313.838, E3 -322678.832}
SPL {X  -142.380, Y  +309.529, Z    +0.000, E1  +319.953, E3 -322751.593}
ENDSPLINE

